IF bComingUp THEN
	IF bEditOffset THEN
		IF bManualPick THEN
			//iCaseRC										:= 900;
			//IF iActualCase = 900 THEN
				bComingUp								:= FALSE;
			//END_IF	
// dodaje druga pozycje pobrania			
		ELSIF bManualPick2 THEN
			//iCaseRC										:= 1600;	
			//IF iActualCase = 1600 THEN
				bComingUp								:= FALSE;
		//	END_IF		
		ELSIF bManualPlace1 THEN
			iCaseRC										:= 1100;	
			IF iActualCase = 1100 THEN
				bComingUp								:= FALSE;
			END_IF	
		ELSIF bManualPlace2 THEN
			iCaseRC										:= 1300;
			//bManualCatch								:= TRUE;
			IF iActualCase = 1300 THEN
				bComingUp								:= FALSE;
			END_IF	
		END_IF	
	ELSE	
		IF iLastCaseRC = 800 THEN												// Pozycja dolna pobierania - komenda
			iCaseRC 										:= 900;
		ELSIF iActualCase = 900 THEN											// Pozycja gorna pobierania - komenda
			iCaseRC											:= 0;
		ELSIF iActualCase = 950 THEN											// Robot w pozycji gornej pobierania
			bComingUp										:= FALSE;
			bManualPick										:= FALSE;			
		ELSIF iLastCaseRC = 1500 THEN											// Pozycja dolna pobierania 2 - komenda
			iCaseRC											:= 1600;
		ELSIF iActualCase = 1600 THEN											// Pozycja gorna pobierania 2 - komenda
			iCaseRC											:= 0;
		ELSIF iActualCase = 1650 THEN											// Robot w pozycji gornej pobierania 2
			bComingUp										:= FALSE;
			bManualPick2									:= FALSE;						
		ELSIF iLastCaseRC = 1000 THEN											// Pozycja dolna odkladania - komenda
			iCaseRC											:= 1100;
		ELSIF iActualCase = 1100 THEN											// Pozycja gorna odkladania - komenda
			iCaseRC											:= 0;
		ELSIF iActualCase = 1150 THEN											// Robot w pozycji gornej odkladania
			bComingUp										:= FALSE;
			bManualPlace1									:= FALSE;
		ELSIF iLastCaseRC = 1200 THEN											// Pozycja dolna odrzutu - komenda
			iCaseRC											:= 1300;
		ELSIF iActualCase = 1300 THEN											// Pozycja gorna odrzutu - komenda
			iCaseRC											:= 0;
		ELSIF iActualCase = 1350 THEN											// Robot w pozycji gornej odrzutu 
			bComingUp										:= FALSE;
			bManualPlace2									:= FALSE;
		END_IF
	END_IF
	iCaseManual												:= 0;	
ELSE
	IF bEditOffset THEN
		IF bManualPick THEN
			iCaseRC											:= 800;				// Pozycja dolna pobierania
		ELSIF bManualPick2 THEN                        	
			iCaseRC											:= 1500;			// Pozycja dolna pobierania 2
		ELSIF bManualPlace1 THEN                        	
			iCaseRC											:= 1000;			// Pozycja dolna odkladanie etykieciarka
		ELSIF bManualPlace2 THEN                        	
			iCaseRC											:= 1200;			// Pozycja dolna odkladania odrzut
		ELSIF iActualCase > 0 THEN                      	
			iCaseRC											:= 0;
		 	bManualPick			:= FALSE;
		 	bManualPick2		:= FALSE;			
		 	bManualPlace1		:= FALSE;
			bManualPlace2		:= FALSE;		
		END_IF	
	iCaseManual												:= 0;	
	ELSE	
//	Case pobranie pojedynczego opakowania	
		IF bManualPick THEN
			CASE iCaseManual OF
				0:
					iCaseRC										:= 200;
					IF iActualCase = 200 THEN
						iCaseRC 								:= 0;
						iCaseManual								:= 10;
					END_IF
				10: 
					IF iActualCase = 250 THEN
						iCaseManual								:= 20;
					END_IF
				20:
					bManualPick									:= FALSE;
					iCaseManual									:= 0;
			END_CASE
		END_IF	
//Dodaje Case bManualPick2 do pobrania dwoch opakowan
		IF bManualPick2 THEN
			CASE iCaseManual OF
				0:
					iCaseRC										:= 1400;
					IF iActualCase = 1400 THEN
						iCaseRC 								:= 0;
						iCaseManual								:= 10;
					END_IF
				10: 
					IF iActualCase = 1450 THEN
						iCaseManual								:= 20;
					END_IF
				20:
					bManualPick2									:= FALSE;
					iCaseManual									:= 0;
			END_CASE
		END_IF		
//	Case odlozenie opakowan na etykieciarke	
		IF bManualPlace1 THEN
			CASE iCaseManual OF
				0:
					iCaseRC										:= 300;
					IF iActualCase = 300 THEN
						iCaseRC 								:= 0;
						iCaseManual								:= 10;
					END_IF
				10: 
					IF iActualCase = 350 THEN
						iCaseManual								:= 20;
					END_IF
				20:
					bManualPlace1								:= FALSE;
					iCaseManual									:= 0;
			END_CASE
		END_IF		
//	Case odlozenie opakowan na odrzut		
		IF bManualPlace2 THEN
			CASE iCaseManual OF
				0:
					iCaseRC										:= 400;
					IF iActualCase = 400 THEN
						iCaseRC 								:= 0;
						iCaseManual								:= 10;
					END_IF
				10: 
					IF iActualCase = 450 THEN
						iCaseManual								:= 20;
					END_IF
				20:
					bManualPlace2								:= FALSE;
					iCaseManual									:= 0;
			END_CASE
		END_IF
//	Case przejazd do pozycji start inkjet		
		IF bManualStartInkJetPosition THEN
			CASE iCaseManual OF
				0:
					iCaseRC										:= 500;
					IF iActualCase = 500 THEN
						iCaseRC 								:= 0;
						iCaseManual								:= 10;
					END_IF
				10: 
					IF iActualCase = 550 THEN
						iCaseManual								:= 20;
					END_IF
				20:
					bManualStartInkJetPosition					:= FALSE;
					iCaseManual									:= 0;
			END_CASE
		END_IF
//	Case przejazd do pozycji stop inkjet		
		IF bManualStopInkJetPosition THEN
			CASE iCaseManual OF
				0:
					iCaseRC										:= 600;
					IF iActualCase = 600 THEN
						iCaseRC 								:= 0;
						iCaseManual								:= 10;
					END_IF
				10: 
					IF iActualCase = 650 THEN
						iCaseManual								:= 20;
					END_IF
				20:
					bManualStopInkJetPosition					:= FALSE;
					iCaseManual									:= 0;
			END_CASE
		END_IF	
		
		IF bManualWeightPosition THEN
			CASE iCaseManual OF
				0:
					iCaseRC										:= 660;
					IF iActualCase = 660 THEN
						iCaseRC 								:= 0;
						iCaseManual								:= 10;
					END_IF
				10: 
					IF iActualCase = 670 THEN
						iCaseManual								:= 20;
					END_IF
				20:	
					iCaseRC										:= 680;
					IF iActualCase = 680 THEN
						iCaseRC 								:= 0;
						iCaseManual								:= 30;
					END_IF	
				30:
					IF iActualCase = 690 THEN
						iCaseManual								:= 40;
					END_IF	
				40:
					bManualWeightPosition						:= FALSE;
					iCaseManual									:= 0;
			END_CASE
		END_IF
		
//	Case przejazd do pozycji gotowosci		
		IF bManualReadyPosition THEN
			CASE iCaseManual OF
				0:
					iCaseRC										:= 700;
					IF iActualCase = 700 THEN
						iCaseRC 								:= 0;
						iCaseManual								:= 10;
					END_IF
				10: 
					IF iActualCase = 750 THEN
						iCaseManual								:= 20;
					END_IF
				20:
					bManualReadyPosition						:= FALSE;
					iCaseManual									:= 0;
			END_CASE
		END_IF	
	END_IF	
END_IF	

IF iCaseRC > 0 THEN
	iLastCaseRC						:= iCaseRC;
END_IF

IF iActualCase=200 OR iActualCase=300 OR iActualCase=400 OR iActualCase=500 OR iActualCase=600 OR iActualCase=700 OR iActualCase=800 OR iActualCase=900 OR iActualCase=1000 OR iActualCase=1100 OR iActualCase=1200 OR iActualCase=1300 OR 
	iActualCase=1400 OR iActualCase=1500 OR iActualCase=1600	THEN
	iBottleTransferLock				:= 2#11111111;	//		nie moge nic
ELSIF iActualCase=150 THEN                                  
	iBottleTransferLock				:= 2#11111110;	//		moge pobrac
ELSIF iActualCase=250 OR iActualCase=950 OR iActualCase=1450 OR iActualCase=1650 THEN	           
	iBottleTransferLock				:= 2#11101001;	//		moge odłozyc, odrzucic i pojechac przed inkjet		
ELSIF iActualCase=350 OR iActualCase=1150 THEN             
	iBottleTransferLock				:= 2#11110111;	//		moge jechac tylko do gotowosci
ELSIF iActualCase=450 OR iActualCase=1350 THEN             
	iBottleTransferLock				:= 2#11110111;	//	   	moge jechac tylko do gotowosci
ELSIF iActualCase=550 THEN                                 
	iBottleTransferLock				:= 2#11011111;	//		moge jechac do koniec inkjet
ELSIF iActualCase=650 THEN                                 
	iBottleTransferLock				:= 2#10101101;	//		moge odłozyc na ety, wrocic przed inkjet
ELSIF iActualCase=750 THEN                                 
	iBottleTransferLock				:= 2#11111110;	//		moge pobrac
END_IF


(*200 pobranie opakowania, 300 odlozenie opakowania, 400 odrzucenie opakowania, 500 przejazd start inkjet, 600 przejazd stop inket, 700 powrot do gotowosci,
800 pozycja dolna pobierania manual, 900 pozycja gorna pobierana manual, 1000 Pozycja dolna odkladania - TRYB MANUALNY, 1100 Pozycja gorna odkladania - TRYB MANUALNY,
1200 Pozycja dolna odrzutu - TRYB MANUALNY, 1300 Pozycja gorna odrzutu - TRYB MANUALNY, 1400 Pobranie  2 opakowan, 1500 Pozycja dolna pobierania 2 - TRYB MANUALNY,
1600 Pozycja gorna pobierania 2 - TRYB MANUALNY


150 - koniec bazowania, 250 - koniec pobierania, 350 - koniec odkladania ety, 450 - koniec odrzutu, 550 - koniec przejazdu do start inket,
650- koniec przejazdu do stop inket, 750 - koniec przejazdu do pozycji gotowosci, 950- koniec gornej pozycji pobrania manual,
1150 - koniec górnej pozycji odkladania manual, 1350 koniec gornej pozycji odrzutu manual, 1450 - koniec pobrania dwoch opakowan,
1650 - koniec gornej pozycji pobrania manual
  *)


(*
IF iActualCase > 0 THEN
	iCaseRC										:= 0;
END_IF
*)
END_ACTION

ACTION Running:
tonWaitForSuckerSensor(IN:=(iActualCase=250 OR iActualCase=350), PT:=T#50MS);

CASE eRunningState OF
  E_RobotMovState.eReadyPlace:	
	iCaseRC								:= 0;
	IF bRun AND NOT bCycleDone THEN
		//Pobór jednego produktu
		IF iPickNumber = 1	THEN
		iCaseRC							:= 200;
			IF iActualCase = 200 THEN
				eRunningState			:= E_RobotMovState.ePicking;
			END_IF
		END_IF
		//Pobor dwóch produktów						
		IF iPickNumber = 2	THEN
		iCaseRC							:= 1400;
			IF iActualCase = 1400 THEN
				eRunningState			:= E_RobotMovState.ePicking;
			END_IF
		END_IF		
		
	END_IF
	
//Sprawdzenie czy poprawnie pobrano produkt
	
	E_RobotMovState.ePicking:
		iCaseRC							:= 0;
		IF  iActualCase = 250 OR iActualLastCase = 250 OR iActualCase = 1450 OR iActualLastCase = 1450 THEN
			iActualLastCase 			:= 0;
			eRunningState				:= E_RobotMovState.ePicked;
		END_IF	

//Sprawdzenie czy popraniw pobrano produkt po zadziałaniu estop	
	E_RobotMovState.ePickingAfterEStop:
		iCaseRC							:= 0;
		IF iActualCase = 280 OR iActualCase = 1480 THEN
			eRunningState				:= E_RobotMovState.ePicked;
		END_IF	
		
// Produkt chwycona do odłożenia 		
	E_RobotMovState.ePicked:
		IF bPlace THEN
			//Odkładanie na etykieciarke
			IF iPlaceNumber = 1 THEN
				IF bInkJetEnable THEN
					iCaseRC				:= 500;
					IF iActualCase = 500 THEN
						eRunningState	:= eMovingInkJetStartPositon;
					END_IF
				ELSE
					iCaseRC				:= 300;
					IF iActualCase = 300 THEN
						eRunningState	:= E_RobotMovState.ePlacing;
					END_IF
				END_IF	
			END_IF
			
			// Odkładanie na odrzut			
			IF iPlaceNumber = 2 THEN
				iCaseRC					:= 400;
				IF iActualCase = 400 THEN
					eRunningState		:= E_RobotMovState.eRejecting;
				END_IF
			END_IF
			
			//Przenoszenie na wagę			
			IF iPlaceNumber = 3 THEN 
				IF bInkJetEnable THEN 
					iCaseRC				:= 500;
					IF iActualCase = 500 THEN
						eRunningState	:= eMovingInkJetStartPositon;
					END_IF
				ELSE
					iCaseRC				:= 660;
					IF iActualCase = 660 THEN
						eRunningState	:= E_RobotMovState.eMovingWeightPosition;
					END_IF
				END_IF	
			END_IF	
			
			
			//Przenoszenie z obrotem
			IF iPlaceNumber = 4 THEN 
				IF bInkJetEnable THEN 
					iCaseRC				:= 500;
					IF iActualCase = 500 THEN
						eRunningState	:= eMovingInkJetStartPositon;
					END_IF
				ELSE
					iCaseRC				:= 1700;
					IF iActualCase = 1700 THEN
						eRunningState	:= E_RobotMovState.eMovingRotatedToPlace;
					END_IF
				END_IF	
			END_IF	
		END_IF		
		
// Sprawdzenie czy odłożono produkt		
	E_RobotMovState.ePlacing:	
		iCaseRC							:= 0;	
		IF iActualCase = 350 THEN
			eRunningState				:= E_RobotMovState.ePlaced;
		END_IF		
		
// Powrót do pozycji gotowości		
	E_RobotMovState.ePlaced:
		iCaseRC							:= 700;
		IF iActualCase = 700 THEN
			eRunningState				:= E_RobotMovState.eReturnToReadyPlace;
		END_IF
		
// Sprawdzenie czy odrzucono produkt		
	E_RobotMovState.eRejecting:
		iCaseRC							:= 0;
		IF iActualCase = 450 THEN	
			eRunningState				:= E_RobotMovState.eRejected;
		END_IF
		
// Sprawdzenie czy odłożono produkt na transporter odrzuconych produktów		
	E_RobotMovState.eRejected:	
		iCaseRC							:= 700;
		IF iActualCase = 700 THEN
			eRunningState				:= E_RobotMovState.eReturnToReadyPlace;
		END_IF
		
// Przejscie do pozycji poczatkowej INKJET		
	E_RobotMovState.eMovingInkJetStartPositon:
		iCaseRC							:= 0;
		IF iActualCase	= 550 THEN
			eRunningState				:= E_RobotMovState.eMovedInkJetStartPositon;
		END_IF
		
// Przejazd INKJET		
	E_RobotMovState.eMovedInkJetStartPositon:
		iCaseRC							:= 600;
		IF iActualCase = 600 THEN
			eRunningState				:= E_RobotMovState.eMovingInkJetStopPositon;
		END_IF	

// Konczenie INJET	
	E_RobotMovState.eMovingInkJetStopPositon:
		iCaseRC							:= 0;	
		IF iActualCase	= 650 THEN
			eRunningState				:= E_RobotMovState.eMovedInkJetStopPositon;
		END_IF	

// Odłożenie opakowania	
	E_RobotMovState.eMovedInkJetStopPositon:
		IF iPlaceNumber = 3 THEN //Przenoszenie na wagę
			iCaseRC				:= 660;
			IF iActualCase = 660 THEN	
				eRunningState	:= eMovingWeightPosition;				
			END_IF 
		ELSE
			iCaseRC							:= 300;	
			IF iActualCase = 300 THEN
				eRunningState				:= E_RobotMovState.ePlacing;
			END_IF	
		END_IF	
	E_RobotMovState.eMovingWeightPosition:
		iCaseRC							:= 0;	
		IF iActualCase = 670 THEN
			eRunningState				:= E_RobotMovState.eMovedWeightPosition;
		END_IF		
	E_RobotMovState.eMovedWeightPosition:
		iCaseRC							:= 680;	
		IF iActualCase = 680 THEN
			eRunningState				:= E_RobotMovState.eMovingAfterWeightPosition;
		END_IF		
	E_RobotMovState.eMovingAfterWeightPosition:
		iCaseRC							:= 0;	
		IF iActualCase = 690 THEN
			eRunningState				:= E_RobotMovState.eMovedAfterWeightPosition;
		END_IF		
	E_RobotMovState.eMovedAfterWeightPosition:
		iCaseRC							:= 300;	
		IF iActualCase = 300 THEN
			eRunningState				:= E_RobotMovState.ePlacing;
		END_IF	
//Odkładanie z obrotem		
	E_RobotMovState.eMovingRotatedToPlace:
		iCaseRC							:= 0;	
		IF iActualCase = 1750 THEN
			eRunningState				:= E_RobotMovState.eReturnToReadyPlace;
		END_IF	
//	E_RobotMovState.eMovedRoatedToPlace:
//		iCaseRC							:= 700;	
//		IF iActualCase = 700 THEN
//			eRunningState				:= E_RobotMovState.eReturnToReadyPlace;
//		END_IF	
		
	
// Konczenie cyklu	
	E_RobotMovState.eReturnToReadyPlace:	
		iCaseRC							:= 0;
		bPlace							:= FALSE;
			//IF iActualCase = 750 THEN
				iLastPickNumber			:= iPlaceNumber;
				bCycleDone				:= TRUE;
			//END_IF
END_CASE

//Tryb wolnych ruchów

IF iPlaceNumber = 1 THEN
	bSlowMotion							:= FALSE;
ELSIF iPlaceNumber = 2 THEN
	bSlowMotion							:= TRUE;	
END_IF
END_ACTION

ACTION Warning:
IF (bEnable) THEN
	
	IF bWarningAcknowledge AND bWarningRCActive  THEN
		bResetWarningRC									:= TRUE;		
	END_IF




	IF bWarningRCActive THEN
		
		bWarning										:= TRUE;
		bWarningNumberRequest							:= TRUE;
		udiWarningId									:= IODATA;
		
		CASE udiWarningId OF	
			
0013:	
	
	sWarningDescription1 := 'Illeagal fileFile Crash';
	sWarningDescription2 := 'File Initial operation';
	
0018:	
	
	sWarningDescription1 := 'The robot model was selected.The robot model was selected.';
	sWarningDescription2 := 'Reset the error';
	
0023:	
	
	sWarningDescription1 := ' Variables save failure (ProgrPower was shutdown before saving program external variables';
	sWarningDescription2 := 'It is necessary to change some parts when not improvement';
	
0024:	
	
	sWarningDescription1 := ' Variables save failure (User)Power was shutdown before saving user-defined external variables';
	sWarningDescription2 := 'The power supply unit might be deteriorated';
	
0029:	
	
	sWarningDescription1 := ' Memory error (ECC)1bit error of ECC was detected';
	sWarningDescription2 := 'When it frequently occurs, contact your service provider';
	
0102:	
	
	sWarningDescription1 := 'Temperature in the Controlle FAN check or Filter at the bottom on Controller becomes old';
	sWarningDescription2 := 'Please exchange the filter to new filter or clean up the filter';
	
0105:	
	
	sWarningDescription1 := ' Temp. in robot CPU is too higAmbient temperature of robot CPU becomes high';
	sWarningDescription2 := 'Please lower ambient temperature to the specification range';
	
0111:	
	
	sWarningDescription1 := ' No UPS battery voltageThe UPS battery is spent';
	sWarningDescription2 := 'Replace the UPS battery';
	
0112:	
	
	sWarningDescription1 := ' Open the UPS battery coverOpen the UPS battery cover';
	sWarningDescription2 := 'Close the UPS battery cover';
	
0114:	
	
	sWarningDescription1 := ' Occur the UPS warningSome abnormalities occurs in UPS';
	sWarningDescription2 := 'Please call S.C.';
	
0120:	
	
	sWarningDescription1 := 'Instantaneous power failureThe power was OFF for 20msec or more';
	sWarningDescription2 := 'Check the power supply connection and power supply state';
	
0150:	
	
	sWarningDescription1 := 'Undefined robot serial numberUndefined robot serial number';
	sWarningDescription2 := 'Input the robot serial number';
	
0151:	
	
	sWarningDescription1 := ' Undefined robot serial numberUndefined robot serial number';
	sWarningDescription2 := 'Input the robot serial number';
	
0152:	
	
	sWarningDescription1 := ' Unmatched robot serial numberRobot arm that connection was replaced';
	sWarningDescription2 := 'Please confirm the connected robot body is not replaced';
	
0190:	
	
	sWarningDescription1 := ' TB not apply present tool No.Connecting TB does not apply present tool number';
	sWarningDescription2 := 'Please operate TB after confirming present tool data(MEXTL)';
	
0200:	
	
	sWarningDescription1 := ' Err.definition file is illegaError number overlapps.';
	sWarningDescription2 := 'Correct Error definition file.';
	
0201:	
	
	sWarningDescription1 := ' Err.definition file is illegaError number is illegal.';
	sWarningDescription2 := 'Correct Error definition file.';
	
0202:	
	
	sWarningDescription1 := ' Err.definition file is illegaError number is out of the range';
	sWarningDescription2 := 'Correct Error definition file.';
	
0203:	
	
	sWarningDescription1 := ' Err.definition file is illegaError definition files form is illegal.';
	sWarningDescription2 := 'Correct Error definition file.';
	
0204:	
	
	sWarningDescription1 := ' Illegal link table was used.System Problem';
	sWarningDescription2 := 'Turn the power OFF and ON once. When it comes back, contact to the dealer.';
	
0205:	
	
	sWarningDescription1 := ' Illegal Error No.System Problem';
	sWarningDescription2 := 'Turn the power OFF and ON once. When it comes back, contact to the dealer.';
	
0240:	
	
	sWarningDescription1 := ' Setting mismatch of safety fuValid/invalid setting of the safety function is a mismatch';
	sWarningDescription2 := 'Turn the power OFF and ON once';
	
0302:	
	
	sWarningDescription1 := ' CR800 test CautionGeneral-purpose Caution for the function test of CR800';
	sWarningDescription2 := 'Check the embedded message';
	
0430:	
	
	sWarningDescription1 := ' Servo amplifier motor overheaThe motor or detectors thermal protector activated';
	sWarningDescription2 := 'Reduce the speed and acceleration of the robot';
	
0460:	
	
	sWarningDescription1 := ' Motor thermal error(Add.Axis)Overheating of the addition axis motor was detected';
	sWarningDescription2 := 'Please exchange the cooling fan of the addition axis motor';
	
1260:	
	
	sWarningDescription1 := 'Encoder communication errorInitial communication error with absolute position linear scale';
	sWarningDescription2 := 'Check the encoder cable connection and conductivity';
	
1270:	
	
	sWarningDescription1 := 'Encoder communication errorThe absolute position serial data was not transmitted correctly';
	sWarningDescription2 := 'Check the encoder cable connection and conductivity';
	
1280:	
	
	sWarningDescription1 := 'Encoder serial format errorAn error was found in the absolute position serial data format';
	sWarningDescription2 := 'Check the encoder cable connection and conductivity';
	
1290:	
	
	sWarningDescription1 := 'Absolute position fluctuationThe absolute position data fluctuated when the power ON';
	sWarningDescription2 := 'Check the axis movement due to arm dropping or external force';
	
1300:	
	
	sWarningDescription1 := 'Servo AMP MP scale F/B errorDeviation was detected in the encoder and MP scale F/B amount';
	sWarningDescription2 := 'Turn the power OFF and ON once';
	
1310:	
	
	sWarningDescription1 := 'Servo AMP MP scale offset errError in the offset data for the ABS position detection system';
	sWarningDescription2 := 'Turn the power OFF and ON once';
	
1320:	
	
	sWarningDescription1 := 'Multi-rotation data errorError was detected in the multi-rotation data for the encoder';
	sWarningDescription2 := 'Turn the power OFF and ON once';
	
1330:	
	
	sWarningDescription1 := 'Encoder battery voltage lowThe voltage of the battery supplying to the encoder has dropped';
	sWarningDescription2 := 'Replace the backup battery';
	
1340:	
	
	sWarningDescription1 := 'Over-regeneration warningThe regeneration level reached 80％ or more';
	sWarningDescription2 := 'Check the load weight or parameter SVPTYP';
	
1350:	
	
	sWarningDescription1 := 'Overload warningThe overload level of servo amplifier reached 80% or more';
	sWarningDescription2 := 'Check the load weight and the robot for collisions, etc';
	
1370:	
	
	sWarningDescription1 := 'Illegal parameter (servo)A parameter was set exceeding the setting range';
	sWarningDescription2 := 'The parameter has not been changed. Reset the correct value';
	
1400:	
	
	sWarningDescription1 := ' regeneration(AUX) frequency oRegeneration at the limit has occurred frequently';
	sWarningDescription2 := 'Check the regeneration capacity';
	
1420:	
	
	sWarningDescription1 := 'Over-regeneration warningThe overload level of converter reached 80% or more';
	sWarningDescription2 := 'Check the load weight or program';
	
1430:	
	
	sWarningDescription1 := 'Servo amplifier main circuit The servo turned ON while the main circuit power was OFF';
	sWarningDescription2 := 'Turn the main circuit power ON';
	
1520:	
	
	sWarningDescription1 := 'Servo motor output watt overThe output wattage of the servo motor exceeded ratings';
	sWarningDescription2 := 'Lower the rotation speed of the servo motor';
	
1580:	
	
	sWarningDescription1 := 'Non-registered servo warningA non-registered servo warning';
	sWarningDescription2 := 'If the warning cannot be reset, turn the power OFF and ON';
	
1620:	
	
	sWarningDescription1 := 'Illegal robot No.The designated robot No. is illegal';
	sWarningDescription2 := 'Set the correct robot No.';
	
1630:	
	
	sWarningDescription1 := 'Cannot servo ON (during errorThe servo cannot be turned ON during a servo error';
	sWarningDescription2 := 'Reset the servo error before turning the servo ON';
	
1650:	
	
	sWarningDescription1 := 'Cannot servo ON (brake OFF)The servo cannot be turned ON when the brakes release';
	sWarningDescription2 := 'Lock the brakes for all axes before turning the servo ON';
	
1660:	
	
	sWarningDescription1 := 'Cannot servo ON (SRVON procesThe servo cannot be turned ON during the servo ON process';
	sWarningDescription2 := 'Do not turn the servo ON during a servo ON process';
	
1670:	
	
	sWarningDescription1 := 'Cannot servo ON (SRVOFF proceThe servo OFF process is being carried out';
	sWarningDescription2 := 'Do not turn the servo OFF during the servo OFF process';
	
1690:	
	
	sWarningDescription1 := 'Cannot brake operation (DEADMThe brakes cannot be released while the DEADMAN switch is OFF';
	sWarningDescription2 := 'Turn the DEADMAN switch ON before operating';
	
1700:	
	
	sWarningDescription1 := 'Cannot brake operation (EMG)The brakes cannot be released while the emergency stop is input';
	sWarningDescription2 := 'Release the emergency stop state before operating';
	
1710:	
	
	sWarningDescription1 := 'Cannot brake operation (SRVONThe brakes cannot be operated during servo ON';
	sWarningDescription2 := 'Turn the servo OFF before operating';
	
1720:	
	
	sWarningDescription1 := 'Cannot brake operation (BRK OThe brakes cannot be released during the brake release process';
	sWarningDescription2 := 'Do not release the brakes during the brake release process';
	
1730:	
	
	sWarningDescription1 := 'Cannot brake operation (BRK OThe brakes cannot be locked during the brake lock process';
	sWarningDescription2 := 'Do not lock the brakes during the brake lock process';
	
1740:	
	
	sWarningDescription1 := 'Servo parameter change failurOther parameter cannot be changed during parameter change';
	sWarningDescription2 := 'Carry out the parameter change process again';
	
1750:	
	
	sWarningDescription1 := 'Servo parameter change failurChanges of the servo parameter failed';
	sWarningDescription2 := 'Carry out the parameter change process again';
	
1760:	
	
	sWarningDescription1 := 'Illegal origin dataThe origin setting data is illegal';
	sWarningDescription2 := 'Set the correct origin data';
	
1761:	
	
	sWarningDescription1 := ' Illegal origin data in robot The origin data is illegal in robot arm';
	sWarningDescription2 := 'Setting the origin';
	
1770:	
	
	sWarningDescription1 := 'Origin setting incompleteThe origin is not set';
	sWarningDescription2 := 'Re-execute after setting the origin';
	
1780:	
	
	sWarningDescription1 := 'Cannot set origin (illegal axThe origin was not set simultaneously for the interference axis';
	sWarningDescription2 := 'Set the origin simultaneously for the interference axis';
	
1781:	
	
	sWarningDescription1 := 'Cannot set origin (SRVON)The origin was set during servo ON';
	sWarningDescription2 := 'Turn the servo OFF before setting the origin';
	
1850:	
	
	sWarningDescription1 := 'Instantaneous power failureThe power was OFF for 20msec or more';
	sWarningDescription2 := 'Check the power supply connection and power supply state';
	
1870:	
	
	sWarningDescription1 := ' Cooling fan stoppedCooling fan in the controller might be out of order';
	sWarningDescription2 := 'Please exchange the cooling fan';
	
1871:	
	
	sWarningDescription1 := 'J1 cooling fan stoppedCooling fan in the controller might be out of order';
	sWarningDescription2 := 'Please exchange the cooling fan';
	
1872:	
	
	sWarningDescription1 := 'J2 cooling fan stoppedCooling fan in the controller might be out of order';
	sWarningDescription2 := 'Please exchange the cooling fan';
	
1873:	
	
	sWarningDescription1 := 'J3 cooling fan stoppedCooling fan in the controller might be out of order';
	sWarningDescription2 := 'Please exchange the cooling fan';
	
1874:	
	
	sWarningDescription1 := 'J4 cooling fan stoppedCooling fan in the controller might be out of order';
	sWarningDescription2 := 'Please exchange the cooling fan';
	
1875:	
	
	sWarningDescription1 := 'J5 cooling fan stoppedCooling fan in the controller might be out of order';
	sWarningDescription2 := 'Please exchange the cooling fan';
	
1876:	
	
	sWarningDescription1 := 'J6 cooling fan stoppedCooling fan in the controller might be out of order';
	sWarningDescription2 := 'Please exchange the cooling fan';
	
1877:	
	
	sWarningDescription1 := 'J7 cooling fan stoppedCooling fan in the controller might be out of order';
	sWarningDescription2 := 'Please exchange the cooling fan';
	
1878:	
	
	sWarningDescription1 := 'J8 cooling fan stoppedCooling fan in the controller might be out of order';
	sWarningDescription2 := 'Please exchange the cooling fan';
	
1890:	
	
	sWarningDescription1 := ' The cooling fan of the additional axis amplifier may be out of order.';
	sWarningDescription2 := '';
	
1891:	
	
	sWarningDescription1 := 'Cooling fan low rev. (add. axCooling fan of the add. axis amp. J1 might be out of order';
	sWarningDescription2 := 'Please exchange the cooling fan';
	
1892:	
	
	sWarningDescription1 := 'Cooling fan low rev. (add. axCooling fan of the add. axis amp. J2 might be out of order';
	sWarningDescription2 := 'Please exchange the cooling fan';
	
1893:	
	
	sWarningDescription1 := 'Cooling fan low rev. (add. axCooling fan of the add. axis amp. J3 might be out of order';
	sWarningDescription2 := 'Please exchange the cooling fan';
	
1894:	
	
	sWarningDescription1 := 'Cooling fan low rev. (add. axCooling fan of the add. axis amp. J4 might be out of order';
	sWarningDescription2 := 'Please exchange the cooling fan';
	
1895:	
	
	sWarningDescription1 := 'Cooling fan low rev. (add. axCooling fan of the add. axis amp. J5 might be out of order';
	sWarningDescription2 := 'Please exchange the cooling fan';
	
1896:	
	
	sWarningDescription1 := 'Cooling fan low rev. (add. axCooling fan of the add. axis amp. J6 might be out of order';
	sWarningDescription2 := 'Please exchange the cooling fan';
	
1897:	
	
	sWarningDescription1 := 'Cooling fan low rev. (add. axCooling fan of the add. axis amp. J7 might be out of order';
	sWarningDescription2 := 'Please exchange the cooling fan';
	
1898:	
	
	sWarningDescription1 := 'Cooling fan low rev. (add. axCooling fan of the add. axis amp. J8 might be out of order';
	sWarningDescription2 := 'Please exchange the cooling fan';
	
1910:	
	
	sWarningDescription1 := 'Cooling fan stopped (amp.)The cooling fan of the servo amp. stopped';
	sWarningDescription2 := 'Confirm the rotation of the servo amp. cooling fan';
	
1920:	
	
	sWarningDescription1 := 'Cooling fan stopped (pow. supThe cooling fan of the power supply stopped';
	sWarningDescription2 := 'Confirm the rotation of the power supply cooling fan';
	
1930:	
	
	sWarningDescription1 := 'Cooling fan stopped (CPU)The cooling fan of the CPU stopped';
	sWarningDescription2 := 'Confirm the rotation of the CPU cooling fan';
	
1940:	
	
	sWarningDescription1 := 'Agitating fan stoppedThe agitating fan in the controller stopped';
	sWarningDescription2 := 'Confirm the rotation of the agitating fan';
	
1960:	
	
	sWarningDescription1 := ' Additional axis AMP warningWarning of the additional axis servo amplifier was detected';
	sWarningDescription2 := 'Please refer to the manual of servo amplifier.';
	
1970:	
	
	sWarningDescription1 := ' Agitating fan stopped (robot)The agitating fan in the robot arm stopped';
	sWarningDescription2 := 'Refer to manual (Troubleshooting)';
	
1990:	
	
	sWarningDescription1 := ' Warning of encoder data errorEncoder positional data error was detected';
	sWarningDescription2 := 'Please check the counter of encoder data error';
	
2040:	
	
	sWarningDescription1 := ' Work coordinate define failedTeaching position is not correct';
	sWarningDescription2 := 'Change the teaching position';
	
2250:	
	
	sWarningDescription1 := ' Safety function is not executSafety function cannot be executed because of origin unsetting';
	sWarningDescription2 := 'Please set the origin';
	
2710:	
	
	sWarningDescription1 := 'CMP error (displacement)The amount of displacement exceeds a regulated value';
	sWarningDescription2 := 'Please reduce displacement';
	
2721:	
	
	sWarningDescription1 := 'CMP error (J1 joint angle)CMP Command exceeds the limit of J1 joint angle';
	sWarningDescription2 := 'Change the position data or reduce displacement';
	
2722:	
	
	sWarningDescription1 := 'CMP error (J2 joint angle)CMP Command exceeds the limit of J2 joint angle';
	sWarningDescription2 := 'Change the position data or reduce displacement';
	
2723:	
	
	sWarningDescription1 := 'CMP error (J3 joint angle)CMP Command exceeds the limit of J3 joint angle';
	sWarningDescription2 := 'Change the position data or reduce displacement';
	
2724:	
	
	sWarningDescription1 := 'CMP error (J4 joint angle)CMP Command exceeds the limit of J4 joint angle';
	sWarningDescription2 := 'Change the position data or reduce displacement';
	
2725:	
	
	sWarningDescription1 := 'CMP error (J5 joint angle)CMP Command exceeds the limit of J5 joint angle';
	sWarningDescription2 := 'Change the position data or reduce displacement';
	
2726:	
	
	sWarningDescription1 := 'CMP error (J6 joint angle)CMP Command exceeds the limit of J6 joint angle';
	sWarningDescription2 := 'Change the position data or reduce displacement';
	
2727:	
	
	sWarningDescription1 := 'CMP error (J7 joint angle)CMP Command exceeds the limit of J7 joint angle';
	sWarningDescription2 := 'Change the position data or reduce displacement';
	
2728:	
	
	sWarningDescription1 := 'CMP error (J8 joint angle)CMP Command exceeds the limit of J8 joint angle';
	sWarningDescription2 := 'Change the position data or reduce displacement';
	
2731:	
	
	sWarningDescription1 := 'CMP error (J1 axis speed)CMP Command exceeds the limit of J1 axis speed';
	sWarningDescription2 := 'Change the position data or reduce the robot motion speed';
	
2732:	
	
	sWarningDescription1 := 'CMP error (J2 axis speed)CMP Command exceeds the limit of J2 axis speed';
	sWarningDescription2 := 'Change the position data or reduce the robot motion speed';
	
2733:	
	
	sWarningDescription1 := 'CMP error (J3 axis speed)CMP Command exceeds the limit of J3 axis speed';
	sWarningDescription2 := 'Change the position data or reduce the robot motion speed';
	
2734:	
	
	sWarningDescription1 := 'CMP error (J4 axis speed)CMP Command exceeds the limit of J4 axis speed';
	sWarningDescription2 := 'Change the position data or reduce the robot motion speed';
	
2735:	
	
	sWarningDescription1 := 'CMP error (J5 axis speed)CMP Command exceeds the limit of J5 axis speed';
	sWarningDescription2 := 'Change the position data or reduce the robot motion speed';
	
2736:	
	
	sWarningDescription1 := 'CMP error (J6 axis speed)CMP Command exceeds the limit of J6 axis speed';
	sWarningDescription2 := 'Change the position data or reduce the robot motion speed';
	
2737:	
	
	sWarningDescription1 := 'CMP error (J7 axis speed)CMP Command exceeds the limit of J7 axis speed';
	sWarningDescription2 := 'Change the position data or reduce the robot motion speed';
	
2738:	
	
	sWarningDescription1 := 'CMP error (J8 axis speed)CMP Command exceeds the limit of J8 axis speed';
	sWarningDescription2 := 'Change the position data or reduce the robot motion speed';
	
2740:	
	
	sWarningDescription1 := 'CMP error (coordinates conv.)CMP Command (POSE type) could not convert to JOINT type';
	sWarningDescription2 := 'Change the position data';
	
2790:	
	
	sWarningDescription1 := ' Cannot teach accurate currentForce control function or CMP command is executed';
	sWarningDescription2 := ' Repeal force control function and compliance mode';
	
3989:	
	
	sWarningDescription1 := ' The test data is undecidedThe tested log data was not decided';
	sWarningDescription2 := 'Please review the argument of the FsTBat command';
	
5610:	
	
	sWarningDescription1 := 'Cannot execute during STOP ONCannot execute during stop signal input';
	sWarningDescription2 := 'Turn the stop signal OFF';
	
5670:	
	
	sWarningDescription1 := ' Cannot execute during waitCannot execute during wait';
	sWarningDescription2 := 'Execute Program Reset';
	
5680:	
	
	sWarningDescription1 := ' Cannot execute while CMP commCannot execute while CMP command is executed';
	sWarningDescription2 := 'Repeal compliance mode (execute CMP OFF)';
	
6050:	
	
	sWarningDescription1 := 'The file cannot be openedMemory size is full';
	sWarningDescription2 := 'Reduce the memory of program size';
	
6060:	
	
	sWarningDescription1 := 'The mode is not TEACHThe mode is not TEACH';
	sWarningDescription2 := 'Carry out parameter writing in the TEACH mode';
	
6070:	
	
	sWarningDescription1 := 'The time cannot be setProgram is runing or robot is SRVON';
	sWarningDescription2 := 'Check the RUN state and that the SRVON state';
	
6080:	
	
	sWarningDescription1 := 'Com mesg is too longCom mesg is too long';
	sWarningDescription2 := 'Check the various settings(ex. Parameters)';
	
6090:	
	
	sWarningDescription1 := 'Can not power reset of robotCan not power reset of robot';
	sWarningDescription2 := 'Can not power reset of robot';
	
6500:	
	
	sWarningDescription1 := 'Not opened COM lineOPEN was not executed by the program';
	sWarningDescription2 := 'Execute OPEN in the program, and then send PRN command';
	
6900:	
	
	sWarningDescription1 := 'Pseudo-input signal modeSet with the parameters';
	sWarningDescription2 := 'When using real signals mode, return the parameter';
	
7000:	
	
	sWarningDescription1 := 'Copy source file was not founThe copy source file was not found';
	sWarningDescription2 := 'Input the correct file name';
	
7010:	
	
	sWarningDescription1 := 'Delete target file was not foThe delete target file was not found';
	sWarningDescription2 := 'Input the correct file name';
	
7020:	
	
	sWarningDescription1 := 'Rename target file was not foThe rename target file was not found';
	sWarningDescription2 := 'Input the correct file name';
	
7040:	
	
	sWarningDescription1 := 'Parameter changes prohibitedChanging this parameter is prohibited as it is dangerous';
	sWarningDescription2 := 'Contact the maker';
	
7070:	
	
	sWarningDescription1 := 'Memory area is fullMemory area is full';
	sWarningDescription2 := 'Delete any unnecessary programs or data';
	
7080:	
	
	sWarningDescription1 := 'Can not read parameterNon-existent parameter or illegal password';
	sWarningDescription2 := '1. Set the correct parameter name. 2. Set the correct password';
	
7081:	
	
	sWarningDescription1 := 'Can not write parameter・Non-existent parameter or illegal password. There are a lot of numbers of characters
							Value is out of range Value is outside the range';
	sWarningDescription2 := '1. Set the correct parameter name. 2. Set the correct password';
	
7082:	
	
	sWarningDescription1 := ' Parameter writing failureFailed in writing the parameter';
	sWarningDescription2 := 'Please confirm a set value and write the parameter again';
	
7090:	
	
	sWarningDescription1 := 'Parameter comment illgalComment illgal';
	sWarningDescription2 := 'Comment is no means.';
	
7110:	
	
	sWarningDescription1 := ' Overhaul period (servo on timThe servo on time has entered the overhaul recommendation period';
	sWarningDescription2 := 'Execution of an overhaul of a robot arm is recommended period';
	
7121:	
	
	sWarningDescription1 := ' Grease replenishment period (Grease consumption degree exceeded the warning level';
	sWarningDescription2 := 'Please replenish grease and reset consumption degree';
	
7122:	
	
	sWarningDescription1 := ' Grease replenishment period (Grease consumption degree exceeded the warning level';
	sWarningDescription2 := 'Please replenish grease and reset consumption degree';
	
7123:	
	
	sWarningDescription1 := ' Grease replenishment period (Grease consumption degree exceeded the warning level';
	sWarningDescription2 := 'Please replenish grease and reset consumption degree';
	
7124:	
	
	sWarningDescription1 := ' Grease replenishment period (Grease consumption degree exceeded the warning level';
	sWarningDescription2 := 'Please replenish grease and reset consumption degree';
	
7125:	
	
	sWarningDescription1 := ' Grease replenishment period (Grease consumption degree exceeded the warning level';
	sWarningDescription2 := 'Please replenish grease and reset consumption degree';
	
7126:	
	
	sWarningDescription1 := ' Grease replenishment period (Grease consumption degree exceeded the warning level';
	sWarningDescription2 := 'Please replenish grease and reset consumption degree';
	
7131:	
	
	sWarningDescription1 := ' Timing belt replacement perioTiming belt consumption degree exceeded the warning level';
	sWarningDescription2 := 'Please replace timing belt and reset consumption degree';
	
7132:	
	
	sWarningDescription1 := ' Timing belt replacement perioTiming belt consumption degree exceeded the warning level';
	sWarningDescription2 := 'Please replace timing belt and reset consumption degree';
	
7133:	
	
	sWarningDescription1 := ' Timing belt replacement perioTiming belt consumption degree exceeded the warning level';
	sWarningDescription2 := 'Please replace timing belt and reset consumption degree';
	
7134:	
	
	sWarningDescription1 := ' Timing belt replacement perioTiming belt consumption degree exceeded the warning level';
	sWarningDescription2 := 'Please replace timing belt and reset consumption degree';
	
7135:	
	
	sWarningDescription1 := ' Timing belt replacement perioTiming belt consumption degree exceeded the warning level';
	sWarningDescription2 := 'Please replace timing belt and reset consumption degree';
	
7136:	
	
	sWarningDescription1 := ' Timing belt replacement perioTiming belt consumption degree exceeded the warning level';
	sWarningDescription2 := 'Please replace timing belt and reset consumption degree';
	
7141:	
	
	sWarningDescription1 := ' Overhaul period (decelerator)Decelerator consumption degree exceeded the warning level';
	sWarningDescription2 := 'Execution of an overhaul of a robot arm is recommended';
	
7142:	
	
	sWarningDescription1 := ' Overhaul period (decelerator)Decelerator consumption degree exceeded the warning level';
	sWarningDescription2 := 'Execution of an overhaul of a robot arm is recommended';
	
7143:	
	
	sWarningDescription1 := ' Overhaul period (decelerator)Decelerator consumption degree exceeded the warning level';
	sWarningDescription2 := 'Execution of an overhaul of a robot arm is recommended';
	
7144:	
	
	sWarningDescription1 := ' Overhaul period (decelerator)Decelerator consumption degree exceeded the warning level';
	sWarningDescription2 := 'Execution of an overhaul of a robot arm is recommended';
	
7145:	
	
	sWarningDescription1 := ' Overhaul period (decelerator)Decelerator consumption degree exceeded the warning level';
	sWarningDescription2 := 'Execution of an overhaul of a robot arm is recommended';
	
7146:	
	
	sWarningDescription1 := ' Overhaul period (decelerator)Decelerator consumption degree exceeded the warning level';
	sWarningDescription2 := 'Execution of an overhaul of a robot arm is recommended';
	
7151:	
	
	sWarningDescription1 := ' Overhaul period (bearing) (J1Bearing consumption degree exceeded the warning level';
	sWarningDescription2 := 'Execution of an overhaul of a robot arm is recommended';
	
7152:	
	
	sWarningDescription1 := ' Overhaul period (bearing) (J2Bearing consumption degree exceeded the warning level';
	sWarningDescription2 := 'Execution of an overhaul of a robot arm is recommended';
	
7153:	
	
	sWarningDescription1 := ' Overhaul period (bearing) (J3Bearing consumption degree exceeded the warning level';
	sWarningDescription2 := 'Execution of an overhaul of a robot arm is recommended';
	
7154:	
	
	sWarningDescription1 := ' Overhaul period (bearing) (J4Bearing consumption degree exceeded the warning level';
	sWarningDescription2 := 'Execution of an overhaul of a robot arm is recommended';
	
7155:	
	
	sWarningDescription1 := ' Overhaul period (bearing) (J5Bearing consumption degree exceeded the warning level';
	sWarningDescription2 := 'Execution of an overhaul of a robot arm is recommended';
	
7156:	
	
	sWarningDescription1 := ' Overhaul period (bearing) (J6Bearing consumption degree exceeded the warning level';
	sWarningDescription2 := 'Execution of an overhaul of a robot arm is recommended';
	
7161:	
	
	sWarningDescription1 := ' Overhaul period (ball screw) Ball screw consumption degree exceeded the war. level';
	sWarningDescription2 := 'Execution of an overhaul of a robot arm is recommended';
	
7162:	
	
	sWarningDescription1 := ' Overhaul period (ball screw) Ball screw consumption degree exceeded the warning level';
	sWarningDescription2 := 'Execution of an overhaul of a robot arm is recommended';
	
7163:	
	
	sWarningDescription1 := ' Overhaul period (ball screw) Ball screw consumption degree exceeded the warning level';
	sWarningDescription2 := 'Execution of an overhaul of a robot arm is recommended';
	
7164:	
	
	sWarningDescription1 := ' Overhaul period (ball screw) Ball screw consumption degree exceeded the warning level';
	sWarningDescription2 := 'Execution of an overhaul of a robot arm is recommended';
	
7165:	
	
	sWarningDescription1 := ' Overhaul period (ball screw) Ball screw consumption degree exceeded the warning level';
	sWarningDescription2 := 'Execution of an overhaul of a robot arm is recommended';
	
7166:	
	
	sWarningDescription1 := ' Overhaul period (ball screw) Ball screw consumption degree exceeded the warning level';
	sWarningDescription2 := 'Execution of an overhaul of a robot arm is recommended';
	
7170:	
	
	sWarningDescription1 := ' Abnormality detection(Dec.)The sign of failure of decelerator was detected';
	sWarningDescription2 := 'Inspection and replacement of decelerator is recommended';
	
7171:	
	
	sWarningDescription1 := ' Abnormality detection(Dec.) (The sign of failure of decelerator was detected';
	sWarningDescription2 := 'Inspection and replacement of decelerator is recommended';
	
7172:	
	
	sWarningDescription1 := ' Abnormality detection(Dec.) (The sign of failure of decelerator was detected';
	sWarningDescription2 := 'Inspection and replacement of decelerator is recommended';
	
7173:	
	
	sWarningDescription1 := ' Abnormality detection(Dec.) (The sign of failure of decelerator was detected';
	sWarningDescription2 := 'Inspection and replacement of decelerator is recommended';
	
7174:	
	
	sWarningDescription1 := ' Abnormality detection(Dec.) (The sign of failure of decelerator was detected';
	sWarningDescription2 := 'Inspection and replacement of decelerator is recommended';
	
7175:	
	
	sWarningDescription1 := ' Abnormality detection(Dec.) (The sign of failure of decelerator was detected';
	sWarningDescription2 := 'Inspection and replacement of decelerator is recommended';
	
7176:	
	
	sWarningDescription1 := ' Abnormality detection(Dec.) (The sign of failure of decelerator was detected';
	sWarningDescription2 := 'Inspection and replacement of decelerator is recommended';
	
7177:	
	
	sWarningDescription1 := ' Abnormality detection(Dec.) (The sign of failure of decelerator was detected';
	sWarningDescription2 := 'Inspection and replacement of decelerator is recommended';
	
7178:	
	
	sWarningDescription1 := ' Abnormality detection(Dec.) (The sign of failure of decelerator was detected';
	sWarningDescription2 := 'Inspection and replacement of decelerator is recommended';
	
7180:	
	
	sWarningDescription1 := ' Abnormality detection(enc datThe sign of failure of encoder was detected';
	sWarningDescription2 := 'Inspection and replacement of motor and wiring is recommended';
	
7181:	
	
	sWarningDescription1 := ' Abnormality detection(enc datThe sign of failure of encoder was detected';
	sWarningDescription2 := 'Inspection and replacement of motor and wiring is recommended';
	
7182:	
	
	sWarningDescription1 := ' Abnormality detection(enc datThe sign of failure of encoder was detected';
	sWarningDescription2 := 'Inspection and replacement of motor and wiring is recommended';
	
7183:	
	
	sWarningDescription1 := ' Abnormality detection(enc datThe sign of failure of encoder was detected';
	sWarningDescription2 := 'Inspection and replacement of motor and wiring is recommended';
	
7184:	
	
	sWarningDescription1 := ' Abnormality detection(enc datThe sign of failure of encoder was detected';
	sWarningDescription2 := 'Inspection and replacement of motor and wiring is recommended';
	
7185:	
	
	sWarningDescription1 := ' Abnormality detection(enc datThe sign of failure of encoder was detected';
	sWarningDescription2 := 'Inspection and replacement of motor and wiring is recommended';
	
7186:	
	
	sWarningDescription1 := ' Abnormality detection(enc datThe sign of failure of encoder was detected';
	sWarningDescription2 := 'Inspection and replacement of motor and wiring is recommended';
	
7187:	
	
	sWarningDescription1 := ' Abnormality detection(enc datThe sign of failure of encoder was detected';
	sWarningDescription2 := 'Inspection and replacement of motor and wiring is recommended';
	
7188:	
	
	sWarningDescription1 := ' Abnormality detection(enc datThe sign of failure of encoder was detected';
	sWarningDescription2 := 'Inspection and replacement of motor and wiring is recommended';
	
7190:	
	
	sWarningDescription1 := ' Abnormality detection(enc comThe sign of failure of encoder was detected';
	sWarningDescription2 := 'Inspection and replacement of motor and wiring is recommended';
	
7191:	
	
	sWarningDescription1 := ' Abnormality detection(enc comThe sign of failure of encoder was detected';
	sWarningDescription2 := 'Inspection and replacement of motor and wiring is recommended';
	
7192:	
	
	sWarningDescription1 := ' Abnormality detection(enc comThe sign of failure of encoder was detected';
	sWarningDescription2 := 'Inspection and replacement of motor and wiring is recommended';
	
7193:	
	
	sWarningDescription1 := ' Abnormality detection(enc comThe sign of failure of encoder was detected';
	sWarningDescription2 := 'Inspection and replacement of motor and wiring is recommended';
	
7194:	
	
	sWarningDescription1 := ' Abnormality detection(enc comThe sign of failure of encoder was detected';
	sWarningDescription2 := 'Inspection and replacement of motor and wiring is recommended';
	
7195:	
	
	sWarningDescription1 := ' Abnormality detection(enc comThe sign of failure of encoder was detected';
	sWarningDescription2 := 'Inspection and replacement of motor and wiring is recommended';
	
7196:	
	
	sWarningDescription1 := ' Abnormality detection(enc comThe sign of failure of encoder was detected';
	sWarningDescription2 := 'Inspection and replacement of motor and wiring is recommended';
	
7197:	
	
	sWarningDescription1 := ' Abnormality detection(enc comThe sign of failure of encoder was detected';
	sWarningDescription2 := 'Inspection and replacement of motor and wiring is recommended';
	
7198:	
	
	sWarningDescription1 := ' Abnormality detection(enc comThe sign of failure of encoder was detected';
	sWarningDescription2 := 'Inspection and replacement of motor and wiring is recommended';
	
7200:	
	
	sWarningDescription1 := ' Add memory has same file.Add memory has file';
	sWarningDescription2 := 'Data clear operation by TB(PROGRAM INIT)';
	
7310:	
	
	sWarningDescription1 := 'Changed variables were not save. The power was OFF during program execution';
	sWarningDescription2 := 'DO NOT turn the power OFF during PROGRAM execution';
	
7320:	
	
	sWarningDescription1 := ' Succeeded in the backup to ROBackup operation was performed';
	sWarningDescription2 := 'As it is, please use it';
	
7321:	
	
	sWarningDescription1 := ' Succeeded in the restore fromAutomatic restoration or compulsive restoration was performed';
	sWarningDescription2 := 'Since ROM data is loaded, please check the contents';
	
7322:	
	
	sWarningDescription1 := ' Failed in the backup to ROMPower supply OFF was carried out during backup processing';
	sWarningDescription2 := 'Please perform backup operation again';
	
7323:	
	
	sWarningDescription1 := ' Failed in the restore from RONone or illegal backup data. or Power supply off of processing';
	sWarningDescription2 := 'Please perform restoration operation again';
	
7324:	
	
	sWarningDescription1 := ' The capacity of ROM and RAM dThere is no extension memory for restoring';
	sWarningDescription2 := 'Please insert an extension memory correctly and perform it again';
	
7410:	
	
	sWarningDescription1 := '1 month inspection is now1 month inspection is now';
	sWarningDescription2 := '1 month inspection is now';
	
7420:	
	
	sWarningDescription1 := '3 month inspection is now3 month inspection is now';
	sWarningDescription2 := '3 month inspection is now';
	
7430:	
	
	sWarningDescription1 := '6 month inspection is now6 month inspection is now';
	sWarningDescription2 := '6 month inspection is now';
	
7440:	
	
	sWarningDescription1 := '1 year inspection is now1 year inspection is now';
	sWarningDescription2 := '1 year inspection is now';
	
7450:	
	
	sWarningDescription1 := 'No battery voltage (robot CPUThe battery is spent';
	sWarningDescription2 := 'Replace the battery and load the data';
	
7451:	
	
	sWarningDescription1 := 'Battery voltage low (robot CPThe battery is spent';
	sWarningDescription2 := 'Replace the battery';
	
7500:	
	
	sWarningDescription1 := 'No battery voltage (robot)The battery is spent';
	sWarningDescription2 := 'Replace the battery and set the origin';
	
7510:	
	
	sWarningDescription1 := 'Battery voltage low (robot)The battery is spent';
	sWarningDescription2 := 'Replace the battery';
	
7520:	
	
	sWarningDescription1 := 'Battery consumption time is oThe battery consumption time was exceeded';
	sWarningDescription2 := 'Replace the battery';
	
7530:	
	
	sWarningDescription1 := 'Replenishment time of greaseIt seems that grease reached longevity';
	sWarningDescription2 := 'Replenish grease';
	
7540:	
	
	sWarningDescription1 := 'Exchange time of the beltIt seems that the belt reached longevity';
	sWarningDescription2 := 'Execute the check and the exchange of the belt';
	
7550:	
	
	sWarningDescription1 := ' Exchange time of the deceleraIt seems that the decelerator reached longevity';
	sWarningDescription2 := 'Execute the check and the exchange of the decelerator';
	
7630:	
	
	sWarningDescription1 := ' No additional-axis cardNo additional-axis card';
	sWarningDescription2 := 'Check additional-axis card';
	
7681:	
	
	sWarningDescription1 := ' Test result was NGThe result of the test processing became NG';
	sWarningDescription2 := 'Please confirm the test object and the test condition';
	
8112:	
	
	sWarningDescription1 := ' ';
	sWarningDescription2 := '';
	
8113:	
	
	sWarningDescription1 := ' ';
	sWarningDescription2 := '';
	
8114:	
	
	sWarningDescription1 := ' ';
	sWarningDescription2 := '';
	
8115:	
	
	sWarningDescription1 := ' ';
	sWarningDescription2 := '';
	
8116:	
	
	sWarningDescription1 := ' ';
	sWarningDescription2 := '';
	
8208:	
	
	sWarningDescription1 := ' There is a possibility of theThe rewriting frequency of ROM exceeded 100000 times';
	sWarningDescription2 := 'Please do not use the trap function';
	
8490:	
	
	sWarningDescription1 := ' DEVICENET Communication test It is communication test mode';
	sWarningDescription2 := 'Please change the mode switch to 3-5 after the test ends';
	
8888:	
	
	sWarningDescription1 := ' Normal Insert-Err MsgNormal Insert-%s-Cause Msg';
	sWarningDescription2 := 'Normal Insert-%s-Measure Msg';
	
8889:	
	
	sWarningDescription1 := ' No InsertMsg-Err MsgNo InsertMsg-Cause Msg';
	sWarningDescription2 := 'No InsertMsg-Measure Msg';
	
8893:	
	
	sWarningDescription1 := ' Get Jiku Nod-Err MsgGet Jiku Nod-Cause Msg';
	sWarningDescription2 := 'Get Jiku Nod Measure Msg';
	
8921:	
	
	sWarningDescription1 := ' Caution of sensor I/F unitThe caution occurred by sensor I/F unit';
	sWarningDescription2 := 'Please refer to the manual of sensor I/F unit';
	
9200:	
	
	sWarningDescription1 := 'User Caution level errorIllegal demand data was transmitted';
	sWarningDescription2 := 'Check program';
	
9201:	
	
	sWarningDescription1 := 'User Caution level errorIllegal demand data was transmitted';
	sWarningDescription2 := 'Check program';
	
9202:	
	
	sWarningDescription1 := 'User Caution level errorIllegal demand data was transmitted';
	sWarningDescription2 := 'Check program';
	
9203:	
	
	sWarningDescription1 := 'User Caution level errorIllegal demand data was transmitted';
	sWarningDescription2 := 'Check program';
	
9204:	
	
	sWarningDescription1 := 'User Caution level errorIllegal demand data was transmitted';
	sWarningDescription2 := 'Check program';
	
9205:	
	
	sWarningDescription1 := 'User Caution level errorIllegal demand data was transmitted';
	sWarningDescription2 := 'Check program';
	
9206:	
	
	sWarningDescription1 := 'User Caution level errorIllegal demand data was transmitted';
	sWarningDescription2 := 'Check program';
	
9207:	
	
	sWarningDescription1 := 'User Caution level errorIllegal demand data was transmitted';
	sWarningDescription2 := 'Check program';
	
9208:	
	
	sWarningDescription1 := 'User Caution level errorIllegal demand data was transmitted';
	sWarningDescription2 := 'Check program';
	
9209:	
	
	sWarningDescription1 := 'User Caution level errorIllegal demand data was transmitted';
	sWarningDescription2 := 'Check program';
	
9210:	
	
	sWarningDescription1 := 'User Caution level errorIllegal demand data was transmitted';
	sWarningDescription2 := 'Check program';
	
9211:	
	
	sWarningDescription1 := 'User Caution level errorIllegal demand data was transmitted';
	sWarningDescription2 := 'Check program';
	
9212:	
	
	sWarningDescription1 := 'User Caution level errorIllegal demand data was transmitted';
	sWarningDescription2 := 'Check program';
	
9213:	
	
	sWarningDescription1 := 'User Caution level errorIllegal demand data was transmitted';
	sWarningDescription2 := 'Check program';
	
9214:	
	
	sWarningDescription1 := 'User Caution level errorIllegal demand data was transmitted';
	sWarningDescription2 := 'Check program';
	
9215:	
	
	sWarningDescription1 := 'User Caution level errorIllegal demand data was transmitted';
	sWarningDescription2 := 'Check program';
	
9216:	
	
	sWarningDescription1 := 'User Caution level errorIllegal demand data was transmitted';
	sWarningDescription2 := 'Check program';
	
9217:	
	
	sWarningDescription1 := 'User Caution level errorIllegal demand data was transmitted';
	sWarningDescription2 := 'Check program';
	
9218:	
	
	sWarningDescription1 := 'User Caution level errorIllegal demand data was transmitted';
	sWarningDescription2 := 'Check program';
	
9219:	
	
	sWarningDescription1 := 'User Caution level errorIllegal demand data was transmitted';
	sWarningDescription2 := 'Check program';
	
9220:	
	
	sWarningDescription1 := 'User Caution level errorIllegal demand data was transmitted';
	sWarningDescription2 := 'Check program';
	
9221:	
	
	sWarningDescription1 := 'User Caution level errorIllegal demand data was transmitted';
	sWarningDescription2 := 'Check program';
	
9222:	
	
	sWarningDescription1 := 'User Caution level errorIllegal demand data was transmitted';
	sWarningDescription2 := 'Check program';
	
9223:	
	
	sWarningDescription1 := 'User Caution level errorIllegal demand data was transmitted';
	sWarningDescription2 := 'Check program';
	
9224:	
	
	sWarningDescription1 := 'User Caution level errorIllegal demand data was transmitted';
	sWarningDescription2 := 'Check program';
	
9225:	
	
	sWarningDescription1 := 'User Caution level errorIllegal demand data was transmitted';
	sWarningDescription2 := 'Check program';
	
9226:	
	
	sWarningDescription1 := 'User Caution level errorIllegal demand data was transmitted';
	sWarningDescription2 := 'Check program';
	
9227:	
	
	sWarningDescription1 := 'User Caution level errorIllegal demand data was transmitted';
	sWarningDescription2 := 'Check program';
	
9228:	
	
	sWarningDescription1 := 'User Caution level errorIllegal demand data was transmitted';
	sWarningDescription2 := 'Check program';
	
9229:	
	
	sWarningDescription1 := 'User Caution level errorIllegal demand data was transmitted';
	sWarningDescription2 := 'Check program';
	
9230:	
	
	sWarningDescription1 := 'User Caution level errorIllegal demand data was transmitted';
	sWarningDescription2 := 'Check program';
	
9231:	
	
	sWarningDescription1 := 'User Caution level errorIllegal demand data was transmitted';
	sWarningDescription2 := 'Check program';
	
9232:	
	
	sWarningDescription1 := 'User Caution level errorIllegal demand data was transmitted';
	sWarningDescription2 := 'Check program';
	
9233:	
	
	sWarningDescription1 := 'User Caution level errorIllegal demand data was transmitted';
	sWarningDescription2 := 'Check program';
	
9234:	
	
	sWarningDescription1 := 'User Caution level errorIllegal demand data was transmitted';
	sWarningDescription2 := 'Check program';
	
9235:	
	
	sWarningDescription1 := 'User Caution level errorIllegal demand data was transmitted';
	sWarningDescription2 := 'Check program';
	
9236:	
	
	sWarningDescription1 := 'User Caution level errorIllegal demand data was transmitted';
	sWarningDescription2 := 'Check program';
	
9237:	
	
	sWarningDescription1 := 'User Caution level errorIllegal demand data was transmitted';
	sWarningDescription2 := 'Check program';
	
9238:	
	
	sWarningDescription1 := 'User Caution level errorIllegal demand data was transmitted';
	sWarningDescription2 := 'Check program';
	
9239:	
	
	sWarningDescription1 := 'User Caution level errorIllegal demand data was transmitted';
	sWarningDescription2 := 'Check program';
	
9240:	
	
	sWarningDescription1 := 'User Caution level errorIllegal demand data was transmitted';
	sWarningDescription2 := 'Check program';
	
9241:	
	
	sWarningDescription1 := 'User Caution level errorIllegal demand data was transmitted';
	sWarningDescription2 := 'Check program';
	
9242:	
	
	sWarningDescription1 := 'User Caution level errorIllegal demand data was transmitted';
	sWarningDescription2 := 'Check program';
	
9243:	
	
	sWarningDescription1 := 'User Caution level errorIllegal demand data was transmitted';
	sWarningDescription2 := 'Check program';
	
9244:	
	
	sWarningDescription1 := 'User Caution level errorIllegal demand data was transmitted';
	sWarningDescription2 := 'Check program';
	
9245:	
	
	sWarningDescription1 := 'User Caution level errorIllegal demand data was transmitted';
	sWarningDescription2 := 'Check program';
	
9246:	
	
	sWarningDescription1 := 'User Caution level errorIllegal demand data was transmitted';
	sWarningDescription2 := 'Check program';
	
9247:	
	
	sWarningDescription1 := 'User Caution level errorIllegal demand data was transmitted';
	sWarningDescription2 := 'Check program';
	
9248:	
	
	sWarningDescription1 := 'User Caution level errorIllegal demand data was transmitted';
	sWarningDescription2 := 'Check program';
	
9249:	
	
	sWarningDescription1 := 'User Caution level errorIllegal demand data was transmitted';
	sWarningDescription2 := 'Check program';
	
9250:	
	
	sWarningDescription1 := 'User Caution level errorIllegal demand data was transmitted';
	sWarningDescription2 := 'Check program';
	
9251:	
	
	sWarningDescription1 := 'User Caution level errorIllegal demand data was transmitted';
	sWarningDescription2 := 'Check program';
	
9252:	
	
	sWarningDescription1 := 'User Caution level errorIllegal demand data was transmitted';
	sWarningDescription2 := 'Check program';
	
9253:	
	
	sWarningDescription1 := 'User Caution level errorIllegal demand data was transmitted';
	sWarningDescription2 := 'Check program';
	
9254:	
	
	sWarningDescription1 := 'User Caution level errorIllegal demand data was transmitted';
	sWarningDescription2 := 'Check program';
	
9255:	
	
	sWarningDescription1 := 'User Caution level errorIllegal demand data was transmitted';
	sWarningDescription2 := 'Check program';
	
9256:	
	
	sWarningDescription1 := 'User Caution level errorIllegal demand data was transmitted';
	sWarningDescription2 := 'Check program';
	
9257:	
	
	sWarningDescription1 := 'User Caution level errorIllegal demand data was transmitted';
	sWarningDescription2 := 'Check program';
	
9258:	
	
	sWarningDescription1 := 'User Caution level errorIllegal demand data was transmitted';
	sWarningDescription2 := 'Check program';
	
9259:	
	
	sWarningDescription1 := 'User Caution level errorIllegal demand data was transmitted';
	sWarningDescription2 := 'Check program';
	
9260:	
	
	sWarningDescription1 := 'User Caution level errorIllegal demand data was transmitted';
	sWarningDescription2 := 'Check program';
	
9261:	
	
	sWarningDescription1 := 'User Caution level errorIllegal demand data was transmitted';
	sWarningDescription2 := 'Check program';
	
9262:	
	
	sWarningDescription1 := 'User Caution level errorIllegal demand data was transmitted';
	sWarningDescription2 := 'Check program';
	
9263:	
	
	sWarningDescription1 := 'User Caution level errorIllegal demand data was transmitted';
	sWarningDescription2 := 'Check program';
	
9264:	
	
	sWarningDescription1 := 'User Caution level errorIllegal demand data was transmitted';
	sWarningDescription2 := 'Check program';
	
9265:	
	
	sWarningDescription1 := 'User Caution level errorIllegal demand data was transmitted';
	sWarningDescription2 := 'Check program';
	
9266:	
	
	sWarningDescription1 := 'User Caution level errorIllegal demand data was transmitted';
	sWarningDescription2 := 'Check program';
	
9267:	
	
	sWarningDescription1 := 'User Caution level errorIllegal demand data was transmitted';
	sWarningDescription2 := 'Check program';
	
9268:	
	
	sWarningDescription1 := 'User Caution level errorIllegal demand data was transmitted';
	sWarningDescription2 := 'Check program';
	
9269:	
	
	sWarningDescription1 := 'User Caution level errorIllegal demand data was transmitted';
	sWarningDescription2 := 'Check program';
	
9270:	
	
	sWarningDescription1 := 'User Caution level errorIllegal demand data was transmitted';
	sWarningDescription2 := 'Check program';
	
9271:	
	
	sWarningDescription1 := 'User Caution level errorIllegal demand data was transmitted';
	sWarningDescription2 := 'Check program';
	
9272:	
	
	sWarningDescription1 := 'User Caution level errorIllegal demand data was transmitted';
	sWarningDescription2 := 'Check program';
	
9273:	
	
	sWarningDescription1 := 'User Caution level errorIllegal demand data was transmitted';
	sWarningDescription2 := 'Check program';
	
9274:	
	
	sWarningDescription1 := 'User Caution level errorIllegal demand data was transmitted';
	sWarningDescription2 := 'Check program';
	
9275:	
	
	sWarningDescription1 := 'User Caution level errorIllegal demand data was transmitted';
	sWarningDescription2 := 'Check program';
	
9276:	
	
	sWarningDescription1 := 'User Caution level errorIllegal demand data was transmitted';
	sWarningDescription2 := 'Check program';
	
9277:	
	
	sWarningDescription1 := 'User Caution level errorIllegal demand data was transmitted';
	sWarningDescription2 := 'Check program';
	
9278:	
	
	sWarningDescription1 := 'User Caution level errorIllegal demand data was transmitted';
	sWarningDescription2 := 'Check program';
	
9279:	
	
	sWarningDescription1 := 'User Caution level errorIllegal demand data was transmitted';
	sWarningDescription2 := 'Check program';
	
9280:	
	
	sWarningDescription1 := 'User Caution level errorIllegal demand data was transmitted';
	sWarningDescription2 := 'Check program';
	
9281:	
	
	sWarningDescription1 := 'User Caution level errorIllegal demand data was transmitted';
	sWarningDescription2 := 'Check program';
	
9282:	
	
	sWarningDescription1 := 'User Caution level errorIllegal demand data was transmitted';
	sWarningDescription2 := 'Check program';
	
9283:	
	
	sWarningDescription1 := 'User Caution level errorIllegal demand data was transmitted';
	sWarningDescription2 := 'Check program';
	
9284:	
	
	sWarningDescription1 := 'User Caution level errorIllegal demand data was transmitted';
	sWarningDescription2 := 'Check program';
	
9285:	
	
	sWarningDescription1 := 'User Caution level errorIllegal demand data was transmitted';
	sWarningDescription2 := 'Check program';
	
9286:	
	
	sWarningDescription1 := 'User Caution level errorIllegal demand data was transmitted';
	sWarningDescription2 := 'Check program';
	
9287:	
	
	sWarningDescription1 := 'User Caution level errorIllegal demand data was transmitted';
	sWarningDescription2 := 'Check program';
	
9288:	
	
	sWarningDescription1 := 'User Caution level errorIllegal demand data was transmitted';
	sWarningDescription2 := 'Check program';
	
9289:	
	
	sWarningDescription1 := 'User Caution level errorIllegal demand data was transmitted';
	sWarningDescription2 := 'Check program';
	
9290:	
	
	sWarningDescription1 := 'User Caution level errorIllegal demand data was transmitted';
	sWarningDescription2 := 'Check program';
	
9291:	
	
	sWarningDescription1 := 'User Caution level errorIllegal demand data was transmitted';
	sWarningDescription2 := 'Check program';
	
9292:	
	
	sWarningDescription1 := 'User Caution level errorIllegal demand data was transmitted';
	sWarningDescription2 := 'Check program';
	
9293:	
	
	sWarningDescription1 := 'User Caution level errorIllegal demand data was transmitted';
	sWarningDescription2 := 'Check program';
	
9294:	
	
	sWarningDescription1 := 'User Caution level errorIllegal demand data was transmitted';
	sWarningDescription2 := 'Check program';
	
9295:	
	
	sWarningDescription1 := 'User Caution level errorIllegal demand data was transmitted';
	sWarningDescription2 := 'Check program';
	
9296:	
	
	sWarningDescription1 := 'User Caution level errorIllegal demand data was transmitted';
	sWarningDescription2 := 'Check program';
	
9297:	
	
	sWarningDescription1 := 'User Caution level errorIllegal demand data was transmitted';
	sWarningDescription2 := 'Check program';
	
9298:	
	
	sWarningDescription1 := 'User Caution level errorIllegal demand data was transmitted';
	sWarningDescription2 := 'Check program';
	
9299:	
	
	sWarningDescription1 := 'User Caution level errorIllegal demand data was transmitted';
	sWarningDescription2 := 'Check program';

			
		END_CASE
		
	ELSE
	bWarningNumberRequest									:= FALSE;
	bResetWarningRC											:= FALSE;	
	bWarning												:= FALSE;
	sWarningDescription1									:= '';
	sWarningDescription2 									:= ''; 
	
	END_IF
	
ELSE
	udiWarningId											:= 0;
	bWarning												:= 	FALSE;
	sWarningDescription1									:= '';
	sWarningDescription2 									:= ''; 
		
END_IF
END_ACTION

END_FUNCTION_BLOCK

// ---- POUs/FB/Conversions/FB_IntTo2Byte.TcPOU
(****************************************************************************************)
(*							Beckhoff Automation Poland									*)
(*								FB_IntTo2Byte	 v1.0									*)
(*									24.5.2011											*)
(*			Blok funkcyjny rozbijający zmienną typu INT na dwie zmienne typu BYTE		*)
(*______________________________________________________________________________________*)
FUNCTION_BLOCK FB_IntTo2Byte
VAR_INPUT
	iInput :INT;
END_VAR
VAR_OUTPUT
	byStarszy : BYTE;
	byMlodszy : BYTE;
END_VAR

byMlodszy := INT_TO_BYTE(iInput);
byStarszy := INT_TO_BYTE(ROL(iInput, 8));

END_FUNCTION_BLOCK

// ---- POUs/P01_TwoPhasesBarriers.TcPOU
PROGRAM P01_TwoPhasesBarriers
VAR_INPUT
IbBarrierBetweenWeightOpenedSensor 			AT %I*: BOOL;	
IbBarrierBetweenWeightClosedSensor 			AT %I*: BOOL;
IbBarrierBetweenDispencerOpenedSensor 		AT %I*: BOOL;
IbBarrierBetweenDispencerClosedSensor 		AT %I*: BOOL;
IbGateBeforeWeights56				 		AT %I*: BOOL;
END_VAR



VAR
	
	QbBarrierBetweenDispencerActuator 			: BOOL; 				 // Wyjście sterujące szlabanem ruchomym pod dozownikami
	//IbBarrierBetweenDispencerOpenedSensor 		AT %I*: BOOL; 			 // Wejście czujnika siłownika środkowej ruchomej bandy pod dozownikami
	//IbBarrierBetweenDispencerClosedSensor 		AT %I*: BOOL; 			 // Wejście czujnika siłownika środkowej ruchomej bandy pod dozownikami

	QbBarrierBetweenWeightActuator 			: BOOL; 				 // Wyjście sterujące szlabanem przed wagami
	
	//IbBarrierBetweenWeightOpenedSensor 			AT %I*: BOOL; 			// Wejście czujnika siłownika środkowej ruchomej bandy przed wjazdem na wagę
	//IbBarrierBetweenWeightClosedSensor 			AT %I*: BOOL; 			// Wejście czujnika siłownika środkowej ruchomej bandy przed wjazdem na wagę

	
	fbBarrierDispencer							: FB_Gate;				// Bloczek obsługi bandy 
	fbBarrierWeight								: FB_Gate;				// Bloczek obsługi bandy 	
	
	bTemp: BOOL;
END_VAR

aBeforeWeight();
aBetweenDispencer();

ACTION aBeforeWeight:
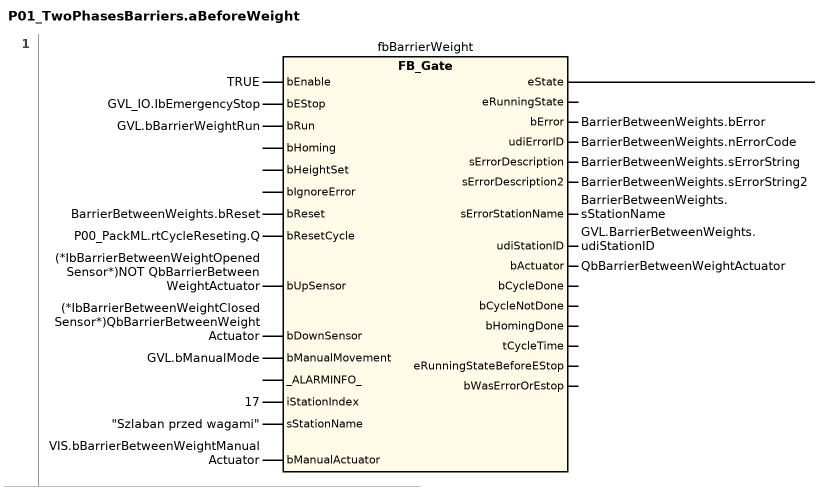
// NETWORK 1
fbBarrierWeight(
    bEnable := TRUE,
    bEStop := GVL_IO.IbEmergencyStop,
    bRun := GVL.bBarrierWeightRun,
    bReset := BarrierBetweenWeights.bReset,
    bResetCycle := P00_PackML.rtCycleReseting.Q,
    bUpSensor := (*IbBarrierBetweenWeightOpenedSensor*)NOT QbBarrierBetweenWeightActuator,
    bDownSensor := (*IbBarrierBetweenWeightClosedSensor*)QbBarrierBetweenWeightActuator,
    bManualMovement := GVL.bManualMode,
    iStationIndex := 17,
    sStationName := "Szlaban przed wagami",
    bManualActuator := VIS.bBarrierBetweenWeightManualActuator,
    bError => BarrierBetweenWeights.bError,
    udiErrorID => BarrierBetweenWeights.nErrorCode,
    sErrorDescription => BarrierBetweenWeights.sErrorString,
    sErrorDescription2 => BarrierBetweenWeights.sErrorString2,
    sErrorStationName => BarrierBetweenWeights.sStationName,
    udiStationID => GVL.BarrierBetweenWeights.udiStationID,
    bActuator => QbBarrierBetweenWeightActuator); // FB_Gate
END_ACTION

ACTION aBetweenDispencer:
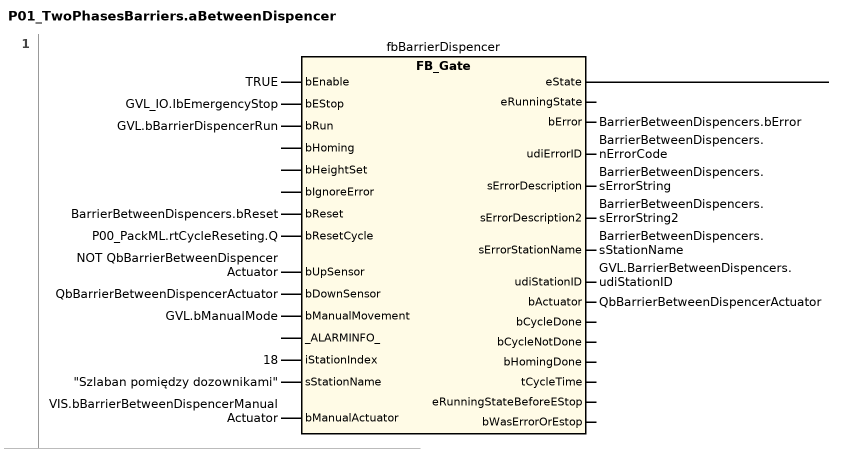
// NETWORK 1
fbBarrierDispencer(
    bEnable := TRUE,
    bEStop := GVL_IO.IbEmergencyStop,
    bRun := GVL.bBarrierDispencerRun,
    bReset := BarrierBetweenDispencers.bReset,
    bResetCycle := P00_PackML.rtCycleReseting.Q,
    bUpSensor := NOT QbBarrierBetweenDispencerActuator,
    bDownSensor := QbBarrierBetweenDispencerActuator,
    bManualMovement := GVL.bManualMode,
    iStationIndex := 18,
    sStationName := "Szlaban pomiędzy dozownikami",
    bManualActuator := VIS.bBarrierBetweenDispencerManualActuator,
    bError => BarrierBetweenDispencers.bError,
    udiErrorID => BarrierBetweenDispencers.nErrorCode,
    sErrorDescription => BarrierBetweenDispencers.sErrorString,
    sErrorDescription2 => BarrierBetweenDispencers.sErrorString2,
    sErrorStationName => BarrierBetweenDispencers.sStationName,
    udiStationID => GVL.BarrierBetweenDispencers.udiStationID,
    bActuator => QbBarrierBetweenDispencerActuator); // FB_Gate
END_ACTION

END_PROGRAM

// ---- POUs/P01_Gates.TcPOU
PROGRAM P01_Gates
VAR_INPUT
	IbGateBeforeWeight14AfterSensor					:BOOL;
	IbLidFeederBarrierOnSensor 	AT %I*  : BOOL;		
    IbLidFeederBarrierOffSensor AT %I*  : BOOL;		
	IbGateBeforeWeights14Sensor	AT %I*	:BOOL;	
	IbGateBeforeWeights56Sensor	AT %I*	:BOOL;		 
END_VAR

VAR
//Szlaban przed dozownikami
	fbGateBeforeDispencers: FB_SpringGateV2;
	fbGateBeforeDispencersState: FB_State;
	eGateBeforeDispencersState :E_Station;
	eGateBeforeDispencersRunningState:E_EntranceGatesState; 
	
	tofTimerGateBeforeDispencersEnable: TOF;
	QbGateBeforeDispencersActuator : BOOL; 				 // Wyjście sterujące szlabanem nr 1 pod robotem
	QbGate0BeforeDispencersActuator : BOOL; 				// Wyjście sterujące szlabanem nr 1 pod robotem
	
//Szlabany przed wagami
	QbGateBeforeWeight14Actuator : BOOL; 			
	QbGateBeforeWeight56Actuator : BOOL; 		

// Szlaban pod stacja robota
	fbGateRobot: FB_SpringGateV2;
	fbGateRobotState: FB_State;
	eGateRobotState :E_Station;
	eGateRobotRunningState:E_EntranceGatesState; 
	tofTimerBottleTransferGatesEnable: TOF;

	QbBottleTransferGate1Actuator : BOOL; 			(*od robota*)	 // Wyjście sterujące szlabanem nr 1 pod robotem
	
	
	fbLidFeederBarrier: FB_Gate;
	QbLidFeederBarrierActuator : BOOL; 	
				
		
	
END_VAR

{warning 'Oprogramować szlaban 0 którego nie było'}
QbGate0BeforeDispencersActuator := QbGateBeforeDispencersActuator;

aGateBeforeDispencers();
aGateBeforeWeight();
aGateRobot();
aLidFeederBarrier();

(***** Generowanie stanu stacji do wizki***********)

//Stan szlabanu przed dozownikami
fbGateBeforeDispencersState(
	eState:= eGateBeforeDispencersState, 
	bRun:=VIS.bGateBeforeDispencersRun AND NOT bManualMode,
	eEntranceGatesRunningState:= eGateBeforeDispencersRunningState, 
	sStateDesc=> VIS.sGateBeforeDispencersState,
	iState=>VIS.iGateBeforeDispencersState);	

(*Opoznienie wyłączanie enabla*)
tofTimerGateBeforeDispencersEnable (IN:=bGateBeforeDispencersEnable , PT:=T#2S);
(*
//Stan szlabanu za wagami
fbGateAfterWeightState(
	eState:= eGateAfterWeightState, 
	bRun:=VIS.bGateAfterWeightEntranceRun AND NOT bManualMode,
	eEntranceGatesRunningState:= eGateAfterWeightRunningState, 
	sStateDesc=> VIS.sGateAfterWeightState,
	iState=>VIS.iGateAfterWeightState);	
*)	
IF P00_PackML.fbPMLAuto.ePMLState = E_PMLState.ePMLState_IDLE THEN
	nGateAfterWeightTimeFormInserting:=250;
END_IF

//Stan szlabanu pod robotem
fbGateRobotState(
	eState:= eGateRobotState, 
	bRun:=VIS.bGateRobotEntranceRun AND NOT bManualMode,
	eEntranceGatesRunningState:= eGateRobotRunningState, 
	sStateDesc=> VIS.sGateRobotState,
	iState=>VIS.iGateRobotState);	
	
IF P00_PackML.fbPMLAuto.ePMLState = E_PMLState.ePMLState_IDLE THEN
	GVL.nGateRobotTimeFormInserting:=250;
END_IF

(*Opoznienie wyłączanie enabla*)
tofTimerBottleTransferGatesEnable (IN:=GVL.bGateRobotEnable , PT:=T#2S);

ACTION aGateBeforeDispencers:
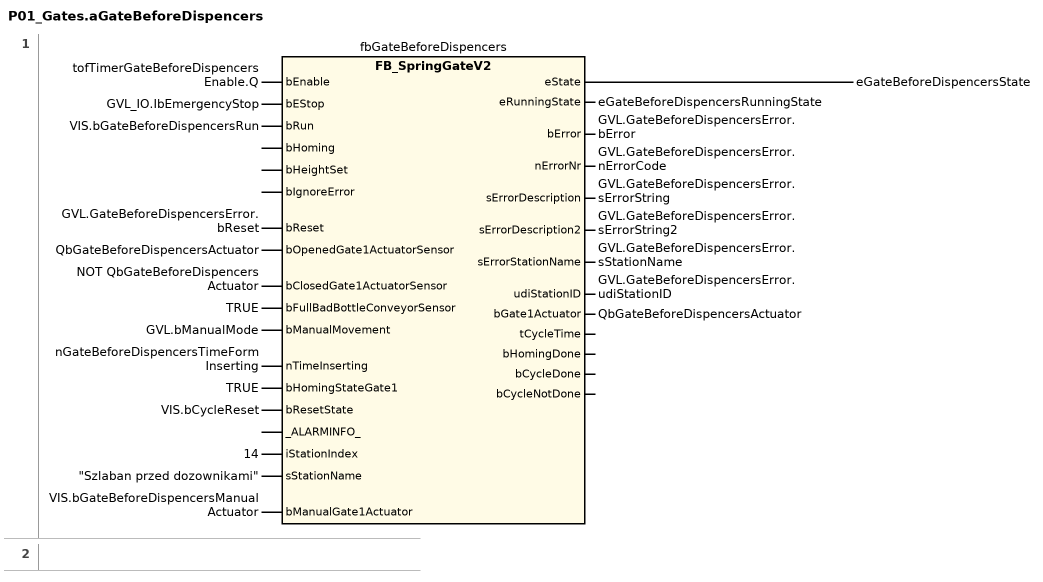
// NETWORK 1
fbGateBeforeDispencers(
    bEnable := tofTimerGateBeforeDispencersEnable.Q,
    bEStop := GVL_IO.IbEmergencyStop,
    bRun := VIS.bGateBeforeDispencersRun,
    bReset := GVL.GateBeforeDispencersError.bReset,
    bOpenedGate1ActuatorSensor := QbGateBeforeDispencersActuator,
    bClosedGate1ActuatorSensor := NOT QbGateBeforeDispencersActuator,
    bFullBadBottleConveyorSensor := TRUE,
    bManualMovement := GVL.bManualMode,
    nTimeInserting := nGateBeforeDispencersTimeFormInserting,
    bHomingStateGate1 := TRUE,
    bResetState := VIS.bCycleReset,
    iStationIndex := 14,
    sStationName := "Szlaban przed dozownikami",
    bManualGate1Actuator := VIS.bGateBeforeDispencersManualActuator,
    eRunningState => eGateBeforeDispencersRunningState,
    bError => GVL.GateBeforeDispencersError.bError,
    nErrorNr => GVL.GateBeforeDispencersError.nErrorCode,
    sErrorDescription => GVL.GateBeforeDispencersError.sErrorString,
    sErrorDescription2 => GVL.GateBeforeDispencersError.sErrorString2,
    sErrorStationName => GVL.GateBeforeDispencersError.sStationName,
    udiStationID => GVL.GateBeforeDispencersError.udiStationID,
    bGate1Actuator => QbGateBeforeDispencersActuator); // FB_SpringGateV2
eGateBeforeDispencersState := fbGateBeforeDispencers.eState;

// NETWORK 2
END_ACTION

ACTION aGateBeforeWeight:

QbGateBeforeWeight14Actuator := VIS.bGateBeforeWeight14Run ;
VIS.bGateBeforeWeight14ManualActuator;

QbGateBeforeWeight56Actuator := VIS.bGateBeforeWeight56Run ;
VIS.bGateBeforeWeight56ManualActuator;
END_ACTION

ACTION aGateRobot:
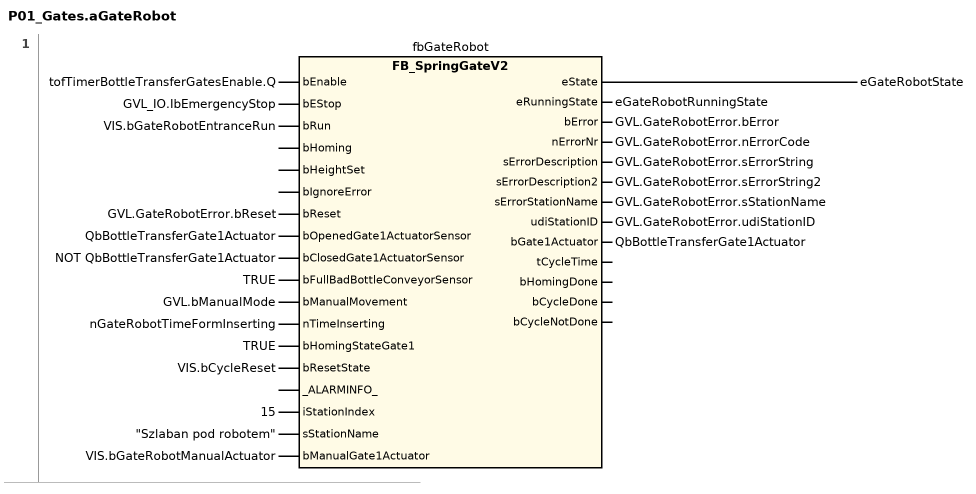
// NETWORK 1
fbGateRobot(
    bEnable := tofTimerBottleTransferGatesEnable.Q,
    bEStop := GVL_IO.IbEmergencyStop,
    bRun := VIS.bGateRobotEntranceRun,
    bReset := GVL.GateRobotError.bReset,
    bOpenedGate1ActuatorSensor := QbBottleTransferGate1Actuator,
    bClosedGate1ActuatorSensor := NOT QbBottleTransferGate1Actuator,
    bFullBadBottleConveyorSensor := TRUE,
    bManualMovement := GVL.bManualMode,
    nTimeInserting := nGateRobotTimeFormInserting,
    bHomingStateGate1 := TRUE,
    bResetState := VIS.bCycleReset,
    iStationIndex := 15,
    sStationName := "Szlaban pod robotem",
    bManualGate1Actuator := VIS.bGateRobotManualActuator,
    eRunningState => eGateRobotRunningState,
    bError => GVL.GateRobotError.bError,
    nErrorNr => GVL.GateRobotError.nErrorCode,
    sErrorDescription => GVL.GateRobotError.sErrorString,
    sErrorDescription2 => GVL.GateRobotError.sErrorString2,
    sErrorStationName => GVL.GateRobotError.sStationName,
    udiStationID => GVL.GateRobotError.udiStationID,
    bGate1Actuator => QbBottleTransferGate1Actuator); // FB_SpringGateV2
eGateRobotState := fbGateRobot.eState;
END_ACTION

ACTION aLidFeederBarrier:
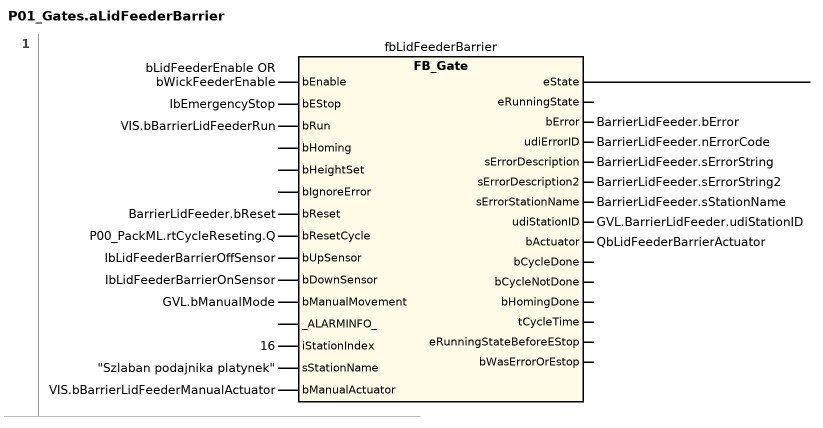
// NETWORK 1
fbLidFeederBarrier(
    bEnable := bLidFeederEnable OR bWickFeederEnable,
    bEStop := IbEmergencyStop,
    bRun := VIS.bBarrierLidFeederRun,
    bReset := BarrierLidFeeder.bReset,
    bResetCycle := P00_PackML.rtCycleReseting.Q,
    bUpSensor := IbLidFeederBarrierOffSensor,
    bDownSensor := IbLidFeederBarrierOnSensor,
    bManualMovement := GVL.bManualMode,
    iStationIndex := 16,
    sStationName := "Szlaban podajnika platynek",
    bManualActuator := VIS.bBarrierLidFeederManualActuator,
    bError => BarrierLidFeeder.bError,
    udiErrorID => BarrierLidFeeder.nErrorCode,
    sErrorDescription => BarrierLidFeeder.sErrorString,
    sErrorDescription2 => BarrierLidFeeder.sErrorString2,
    sErrorStationName => BarrierLidFeeder.sStationName,
    udiStationID => GVL.BarrierLidFeeder.udiStationID,
    bActuator => QbLidFeederBarrierActuator); // FB_Gate
END_ACTION

END_PROGRAM

// ---- POUs/P05_Weight.TcPOU
(*
Nazwa:			P05_Weight
Opis:			Stacja wagi
Wersja:			v0.2
Data:			2019-10-1
Autor:			DP
Urzadzenia:		
Konfiguracja:	
Info:
-przerobione na wagę beckhofa
*)
PROGRAM P05_Weight
VAR_INPUT
	IbWeight1FormSensor						AT %I*		: BOOL;							//Czujnik nad Waga 1
	IbWeight2FormSensor						AT %I*		: BOOL;							//Czujnik nad Waga 2
	IbWeight3FormSensor						AT %I*		: BOOL;							//Czujnik nad Waga 3
	IbWeight4FormSensor						AT %I*		: BOOL;							//Czujnik nad Waga 4
	IbWeight5FormSensor						AT %I*		: BOOL;							//Czujnik nad Waga 4
	IbWeight6FormSensor						AT %I*		: BOOL;							//Czujnik nad Waga 4
END_VAR
VAR
	//Podnosnik szalek
	
	//eWeightLiftRunningState			:E_WeightLiftState;				// Stan pracy podajnika
	fbWeightLiftState					:FB_State;
	
	//Waga 1
	fbWeight1							:FB_BeckhoffEL3356Weight;		// Blok sterujący pierwszą wagą
	eWeight1State						:E_Station; 					// Stan pracy podajnika platynek			
	eWeight1RunningState				:E_WeightState; 				// Stan pracy podajnika platynek
	fbWeight1State						:FB_State;					

	(*No nowej wagi*)
	(*wejścia*)
	InWeight1Value						 AT %I*: DINT;			// Wartość wagi
	IbWeight1Overrange					 AT %I*: BOOL;						
	IbWeight1DataInvalid				 AT %I*: BOOL;		
	IbWeight1Error 						 AT %I*: BOOL;	
	IbWeight1CalibrationInProgress 		 AT %I*: BOOL;
	IbWeight1SteadyState				 AT %I*: BOOL;
	IbWeight1SyncError 					 AT %I*: BOOL;
	(*wyjścia*)
	QbWeight1StartCalibration 			 AT %Q*: BOOL;
	QbWeight1DisableCalibration     	 AT %Q*: BOOL;
	QbWeight1InputFreeze 				 AT %Q*: BOOL;
	QbWeight1SampleMode 				 AT %Q*: BOOL;
	QbWeight1Tara 					     AT %Q*: BOOL;
	
	(*Ostrzezenia*)
	bWeight1Warning1					:BOOL; // 
	tonWeight1Tare						:TON;
	
	//Waga 2
	fbWeight2							:FB_BeckhoffEL3356Weight;		// Blok sterujący pierwszą wagą
	eWeight2State						:E_Station; 					// Stan pracy podajnika platynek			
	eWeight2RunningState				:E_WeightState; 				// Stan pracy podajnika platynek
	fbWeight2State						:FB_State;					

	(*No nowej wagi*)
	(*wejścia*)
	InWeight2Value 						AT %I*: DINT;			// Wartość wagi
	IbWeight2Overrange 					AT %I*: BOOL;						
	IbWeight2DataInvalid 				AT %I*: BOOL;		
	IbWeight2Error 						AT %I*: BOOL;	
	IbWeight2CalibrationInProgress		AT %I*: BOOL;
	IbWeight2SteadyState 				AT %I*: BOOL;
	IbWeight2SyncError 					AT %I*: BOOL;
	(*wyjścia*)
	QbWeight2StartCalibration 			AT %Q*: BOOL;
	QbWeight2DisableCalibration			AT %Q*: BOOL;
	QbWeight2InputFreeze 				AT %Q*: BOOL;
	QbWeight2SampleMode 				AT %Q*: BOOL;
	QbWeight2Tara 						AT %Q*: BOOL;
	
	(*Ostrzezenia*)
	bWeight2Warning1					:BOOL; // 
	tonWeight2Tare						:TON;
		
	//Waga 3
	fbWeight3							:FB_BeckhoffEL3356Weight;		// Blok sterujący pierwszą wagą
	eWeight3State						:E_Station; 					// Stan pracy podajnika platynek			
	eWeight3RunningState				:E_WeightState; 				// Stan pracy podajnika platynek
	fbWeight3State						:FB_State;					

	(*No nowej wagi*)
	(*wejścia*)
	InWeight3Value						 AT %I*: DINT;			// Wartość wagi
	IbWeight3Overrange 					 AT %I*: BOOL;						
	IbWeight3DataInvalid 				 AT %I*: BOOL;		
	IbWeight3Error 						 AT %I*: BOOL;	
	IbWeight3CalibrationInProgress 		 AT %I*: BOOL;
	IbWeight3SteadyState 				 AT %I*: BOOL;
	IbWeight3SyncError 					 AT %I*: BOOL;
	(*wyjścia*)
	QbWeight3StartCalibration 			 AT %Q*: BOOL;
	QbWeight3DisableCalibration 		 AT %Q*: BOOL;
	QbWeight3InputFreeze 				 AT %Q*: BOOL;
	QbWeight3SampleMode 			   	 AT %Q*: BOOL;
	QbWeight3Tara 						 AT %Q*: BOOL;
	
	(*Ostrzezenia*)
	bWeight3Warning1					:BOOL; // 
	tonWeight3Tare						: TON;	
	
	//Waga 4
	fbWeight4							:FB_BeckhoffEL3356Weight;		// Blok sterujący pierwszą wagą
	eWeight4State						:E_Station; 					// Stan pracy podajnika platynek			
	eWeight4RunningState				:E_WeightState; 				// Stan pracy podajnika platynek
	fbWeight4State						:FB_State;					

	(*No nowej wagi*)
	(*wejścia*)
	InWeight4Value 						AT %I*: DINT;			// Wartość wagi
	IbWeight4Overrange 					AT %I*: BOOL;						
	IbWeight4DataInvalid				AT %I*: BOOL;		
	IbWeight4Error 						AT %I*: BOOL;	
	IbWeight4CalibrationInProgress 		AT %I*: BOOL;
	IbWeight4SteadyState 				AT %I*: BOOL;
	IbWeight4SyncError 					AT %I*: BOOL;
	(*wyjścia*)
	QbWeight4StartCalibration 			AT %Q*: BOOL;
	QbWeight4DisableCalibration 		AT %Q*: BOOL;
	QbWeight4InputFreeze 				AT %Q*: BOOL;
	QbWeight4SampleMode 				AT %Q*: BOOL;
	QbWeight4Tara 						AT %Q*: BOOL;

	(*Ostrzezenia*)
	bWeight4Warning1					:BOOL; // 
	tonWeight4Tare						:TON;	
		
(******** Dozowanie dwufazowe******)	
////// Wagi przy dozowaniu dwufazowym dodano 07.04.2022
	//Waga 5
	fbWeight5							:FB_BeckhoffEL3356Weight;		// Blok sterujący pierwszą wagą
	eWeight5State						:E_Station; 					// Stan pracy podajnika platynek			
	eWeight5RunningState				:E_WeightState; 				// Stan pracy podajnika platynek
	fbWeight5State						:FB_State;					

	(*No nowej wagi*)
	(*wejścia*)
	InWeight5Value 						AT %I*: DINT;			// Wartość wagi
	IbWeight5Overrange 					AT %I*: BOOL;						
	IbWeight5DataInvalid 				AT %I*: BOOL;		
	IbWeight5Error 						AT %I*: BOOL;	
	IbWeight5CalibrationInProgress 		AT %I*: BOOL;
	IbWeight5SteadyState 				AT %I*: BOOL;
	IbWeight5SyncError 					AT %I*: BOOL;
	(*wyjścia*)
	QbWeight5StartCalibration 			AT %Q*: BOOL;
	QbWeight5DisableCalibration 		AT %Q*: BOOL;
	QbWeight5InputFreeze 				AT %Q*: BOOL;
	QbWeight5SampleMode 				AT %Q*: BOOL;
	QbWeight5Tara 						AT %Q*: BOOL;

	(*Ostrzezenia*)
	bWeight5Warning1					:BOOL; // 
	tonWeight5Tare						:TON;		
	
	//Waga 5
	fbWeight6							:FB_BeckhoffEL3356Weight;		// Blok sterujący pierwszą wagą
	eWeight6State						:E_Station; 					// Stan pracy podajnika platynek			
	eWeight6RunningState				:E_WeightState; 				// Stan pracy podajnika platynek
	fbWeight6State						:FB_State;					

	(*No nowej wagi*)
	(*wejścia*)
	InWeight6Value 						AT %I*: DINT;			// Wartość wagi
	IbWeight6Overrange 					AT %I*: BOOL;						
	IbWeight6DataInvalid 				AT %I*: BOOL;		
	IbWeight6Error 						AT %I*: BOOL;	
	IbWeight6CalibrationInProgress 		AT %I*: BOOL;
	IbWeight6SteadyState 				AT %I*: BOOL;
	IbWeight6SyncError 					AT %I*: BOOL;
	(*wyjścia*)
	QbWeight6StartCalibration 			AT %Q*: BOOL;
	QbWeight6DisableCalibration 		AT %Q*: BOOL;
	QbWeight6InputFreeze 				AT %Q*: BOOL;
	QbWeight6SampleMode 				AT %Q*: BOOL;
	QbWeight6Tara 						AT %Q*: BOOL;

	(*Ostrzezenia*)
	bWeight6Warning1					:BOOL; // 
	tonWeight6Tare						:TON;		
	
(******** Dozowanie dwufazowe******)		
	
	//Czujniki optyczne przed i za wagą
	fbFilterWeight1: FB_FilterEx;
	fbFilterWeight2: FB_FilterEx;
	fbFilterWeight3: FB_FilterEx;
	fbFilterWeight4: FB_FilterEx;
	fbFilterWeight5: FB_FilterEx;(****** dodane 07.04.2022 przy dodzowniu dwufazowym	**)
	fbFilterWeight6: FB_FilterEx;(****** dodane 07.04.2022 przy dodzowniu dwufazowym	**)

	rFilteredWeight1Value: REAL;
	rFilteredWeight2Value: REAL;
	rFilteredWeight3Value: REAL;
	rFilteredWeight4Value: REAL;
	rFilteredWeight5Value: REAL;(****** dodane 07.04.2022 przy dodzowniu dwufazowym	**)
	rFilteredWeight6Value: REAL;(****** dodane 07.04.2022 przy dodzowniu dwufazowym	**)
	
	//Damian dodane 2 fazy
	fbWeightStation2Phase							: FB_WeightStation;	
	eWeightStation2PhaseState						: E_Station;
	eWeightStation2PhaseRunningState				: E_WeightLiftStationState;
	
	//Dodane Przez Mikołaja
	fbWeightStation									: FB_WeightStation;
	eWeightStationState								: E_Station;
	eWeightStationRunningState						: E_WeightLiftStationState;
	
	IbWeight1ActuatorSensorUp			AT %I*		: BOOL;							//Czujnik podnoszenia Waga 1
	IbWeight2ActuatorSensorUp			AT %I*		: BOOL;							//Czujnik podnoszenia Waga 2
	IbWeight3ActuatorSensorUp			AT %I*		: BOOL;							//Czujnik podnoszenia Waga 3
	IbWeight4ActuatorSensorUp			AT %I*		: BOOL;							//Czujnik podnoszenia Waga 4
	IbWeight5ActuatorSensorUp			AT %I*		: BOOL;							//Czujnik podnoszenia Waga 5 
	IbWeight6ActuatorSensorUp			AT %I*		: BOOL;							//Czujnik podnoszenia Waga 6 
		
	QbWeight1Actuator								: BOOL;							//Podnoszenie Waga 1
    QbWeight2Actuator								: BOOL;							//Podnoszenie Waga 2
	QbWeight3Actuator								: BOOL;							//Podnoszenie Waga 3
	QbWeight4Actuator								: BOOL;							//Podnoszenie Waga 4	                                    		
	QbWeight5Actuator								: BOOL;							//Podnoszenie Waga 5 (2faza)	                                    		
	QbWeight6Actuator								: BOOL;							//Podnoszenie Waga 6 (2faza)

		
	(*Symulacja czujników*)
	tonIbWeight1ActuatorSensorUp					: TON;	
	tonIbWeight2ActuatorSensorUp					: TON;	
	tonIbWeight3ActuatorSensorUp					: TON;	
	tonIbWeight4ActuatorSensorUp					: TON;	
	tonIbWeight5ActuatorSensorUp					: TON;	
	tonIbWeight6ActuatorSensorUp					: TON;	
	
	tonIbWeight1FormSensor: TON;
	tonIbWeight2FormSensor: TON;
	tonIbWeight3FormSensor: TON;
	tonIbWeight4FormSensor: TON;
	tonIbWeight5FormSensor: TON;
	tonIbWeight6FormSensor: TON;
	
	fbIbWeight1FormBeforeSensor: FB_InputFilter_v2;
	fbIbWeight2FormBeforeSensor: FB_InputFilter_v2;
	fbIbWeight3FormBeforeSensor: FB_InputFilter_v2;
	fbIbWeight4FormBeforeSensor: FB_InputFilter_v2;		
	fbIbWeight5FormBeforeSensor: FB_InputFilter_v2;		
	fbIbWeight6FormBeforeSensor: FB_InputFilter_v2;			
	btemp: BOOL;
	
	//wykresy
	fbTrig1 : R_TRIG;
    fbTrig2 : R_TRIG;
    fbTrig3 : R_TRIG;
    fbTrig4 : R_TRIG;
	tSys : DT;
    tTOD : TOD;
	GetTimeSeconds : INT;
	weightIndex : INT;   // 0..7
    valueY : INT;
	i : INT;
	 
	fbHistory: FB_WeightHistory;
END_VAR


fbWeight1.bIgnoreError:=fbWeight2.bIgnoreError:=fbWeight3.bIgnoreError:=fbWeight4.bIgnoreError:=fbWeight5.bIgnoreError:=fbWeight6.bIgnoreError;

aFilter();
aWeight1();
aWeight2();
aWeight3();
aWeight4();
aWeight5();
aWeight6();
ACT_WeightChartDrawers();
IF NOT bDosingTwoPhases THEN
	ACT_WeightStation();
ELSE
	ACT_WeightStation2Phase();
END_IF

// Czas opóżnienia zbierania próbekFB_EntranceGatesServo
fbWeight1.nWeightingDelay:=fbWeight2.nWeightingDelay:=fbWeight3.nWeightingDelay:=fbWeight4.nWeightingDelay:=530;//530
fbWeight5.nWeightingDelay:=fbWeight6.nWeightingDelay:=750;//było 685

(********* GENEROWANIE STANU STACJI DO WIZKI**********)

fbWeight1State(
	eState															:= eWeight1State , 
	bRun															:= VIS.bWeight1DoWeighting,	
	eWeightRunningState												:= eWeight1RunningState , 
	sStateDesc														=> VIS.sWeight1State,
	iState															=> VIS.iWeight1State	);	

fbWeight2State(
	eState															:= eWeight2State , 
	bRun															:= VIS.bWeight2DoWeighting,	
	eWeightRunningState												:= eWeight2RunningState , 
	sStateDesc														=> VIS.sWeight2State,
	iState															=> VIS.iWeight2State	);	
		
fbWeight3State(
	eState															:= eWeight3State , 
	bRun															:= VIS.bWeight3DoWeighting,	
	eWeightRunningState												:= eWeight3RunningState , 
	sStateDesc														=> VIS.sWeight3State,
	iState															=> VIS.iWeight3State	);	
	
fbWeight4State(
	eState															:= eWeight4State , 
	bRun															:= VIS.bWeight4DoWeighting,	
	eWeightRunningState												:= eWeight4RunningState , 
	sStateDesc														=> VIS.sWeight4State,
	iState															=> VIS.iWeight4State	);	
	
fbWeight5State(
	eState															:= eWeight5State , 
	bRun															:= VIS.bWeight5DoWeighting,	
	eWeightRunningState												:= eWeight5RunningState , 
	sStateDesc														=> VIS.sWeight5State,
	iState															=> VIS.iWeight5State	);	

fbWeight6State(
	eState															:= eWeight6State , 
	bRun															:= VIS.bWeight6DoWeighting,	
	eWeightRunningState												:= eWeight6RunningState , 
	sStateDesc														=> VIS.sWeight6State,
	iState															=> VIS.iWeight6State	);		
	
fbWeightLiftState(
	eState															:= eWeightStationState, 
	bRun															:= VIS.bWeightLiftRun OR bWeightLift2PhaseRun,	
	eWeightLiftRunningState											:= eWeightStationRunningState , 
	sStateDesc														=> VIS.sWeightLiftState,
	iState															=> VIS.iWeightLiftState	);		
	
(***** KONIEC GENEROWANIE STANU STACJI DO WIZKI*******)

(****Ostrzezenia***)
// Waga 1
WeightWarning[0].sDescription										:= 'Wagi | Brak stabilizacji przy pomiarach';
IF (bWeight1Warning1 OR bWeight2Warning1 OR bWeight3Warning1 OR bWeight4Warning1 OR bWeight5Warning1 OR bWeight6Warning1) AND NOT WeightWarning[0].bWarning THEN
	WeightWarning[0].bWarning										:= TRUE;
	
ELSIF NOT bWeight1Warning1 AND WeightWarning[0].bAcknowledge THEN
	WeightWarning[0].bWarning										:= FALSE;
	WeightWarning[0].bAcknowledge									:= FALSE;
	VIS.uliWarningAcknowledge.4 										:= FALSE;
	
ELSIF WeightWarning[0].bAcknowledge THEN
	WeightWarning[0].bAcknowledge									:= TRUE;
END_IF


(********KASOWANIE ROZKAZÓW CYKLI*********)
IF fbWeight1.bCycleDone AND bManualMode THEN
	VIS.bWeight1DoWeighting 												:= FALSE;
END_IF

tonWeight1Tare(IN:=VIS.bWeight1Tare,PT:=T#2S);
IF tonWeight1Tare.Q THEN
	VIS.bWeight1Tare												:= FALSE;
END_IF

IF fbWeight2.bCycleDone AND bManualMode THEN
	VIS.bWeight2DoWeighting 												:= FALSE;
END_IF

tonWeight2Tare(IN:=VIS.bWeight2Tare,PT:=T#2S);
IF tonWeight2Tare.Q THEN
	VIS.bWeight2Tare												:= FALSE;
END_IF

IF fbWeight3.bCycleDone AND bManualMode THEN
	VIS.bWeight3DoWeighting 												:= FALSE;
END_IF

tonWeight3Tare(IN:=VIS.bWeight3Tare,PT:=T#2S);
IF tonWeight3Tare.Q THEN
	VIS.bWeight3Tare												:= FALSE;
END_IF
//
IF fbWeight4.bCycleDone AND bManualMode THEN
	VIS.bWeight4DoWeighting 												:= FALSE;
END_IF

tonWeight4Tare(IN:=VIS.bWeight4Tare,PT:=T#2S);
IF tonWeight4Tare.Q THEN
	VIS.bWeight4Tare												:= FALSE;
END_IF

// Waga 5 (1 stacja przy dwufazie)
IF fbWeight5.bCycleDone AND bManualMode THEN
	VIS.bWeight5DoWeighting 												:= FALSE;
END_IF

tonWeight5Tare(IN:=VIS.bWeight5Tare,PT:=T#2S);
IF tonWeight5Tare.Q THEN
	VIS.bWeight5Tare												:= FALSE;
END_IF

// Waga 6 (1 stacja przy dwufazie)
IF fbWeight6.bCycleDone AND bManualMode THEN
	VIS.bWeight6DoWeighting 												:= FALSE;
END_IF

tonWeight6Tare(IN:=VIS.bWeight6Tare,PT:=T#2S);
IF tonWeight6Tare.Q THEN
	VIS.bWeight6Tare												:= FALSE;
END_IF
(*****KONIEC KASOWANIA ROZKAZÓW CYKLI*****)

(**SYMULACJA CZUJNIKÓW**)
tonIbWeight1ActuatorSensorUp(IN:= QbWeight1Actuator, PT:=T#80MS);
tonIbWeight2ActuatorSensorUp(IN:= QbWeight2Actuator, PT:=T#80MS);
tonIbWeight3ActuatorSensorUp(IN:= QbWeight3Actuator, PT:=T#80MS);
tonIbWeight4ActuatorSensorUp(IN:= QbWeight4Actuator, PT:=T#80MS);
tonIbWeight5ActuatorSensorUp(IN:= QbWeight5Actuator, PT:=T#100MS);
tonIbWeight6ActuatorSensorUp(IN:= QbWeight6Actuator, PT:=T#100MS);

ACTION ACT_WeightChartDrawers:
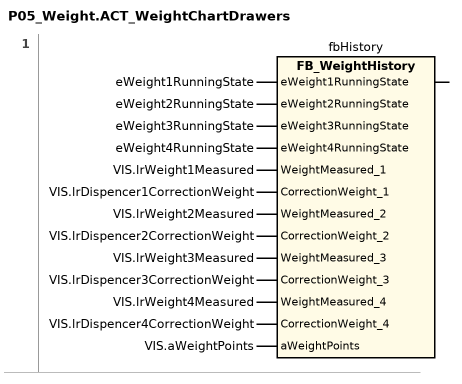
// NETWORK 1
fbHistory(
    eWeight1RunningState := eWeight1RunningState,
    eWeight2RunningState := eWeight2RunningState,
    eWeight3RunningState := eWeight3RunningState,
    eWeight4RunningState := eWeight4RunningState,
    WeightMeasured_1 := VIS.lrWeight1Measured,
    CorrectionWeight_1 := VIS.lrDispencer1CorrectionWeight,
    WeightMeasured_2 := VIS.lrWeight2Measured,
    CorrectionWeight_2 := VIS.lrDispencer2CorrectionWeight,
    WeightMeasured_3 := VIS.lrWeight3Measured,
    CorrectionWeight_3 := VIS.lrDispencer3CorrectionWeight,
    WeightMeasured_4 := VIS.lrWeight4Measured,
    CorrectionWeight_4 := VIS.lrDispencer4CorrectionWeight,
    aWeightPoints := VIS.aWeightPoints); // FB_WeightHistory
END_ACTION

ACTION ACT_WeightStation:
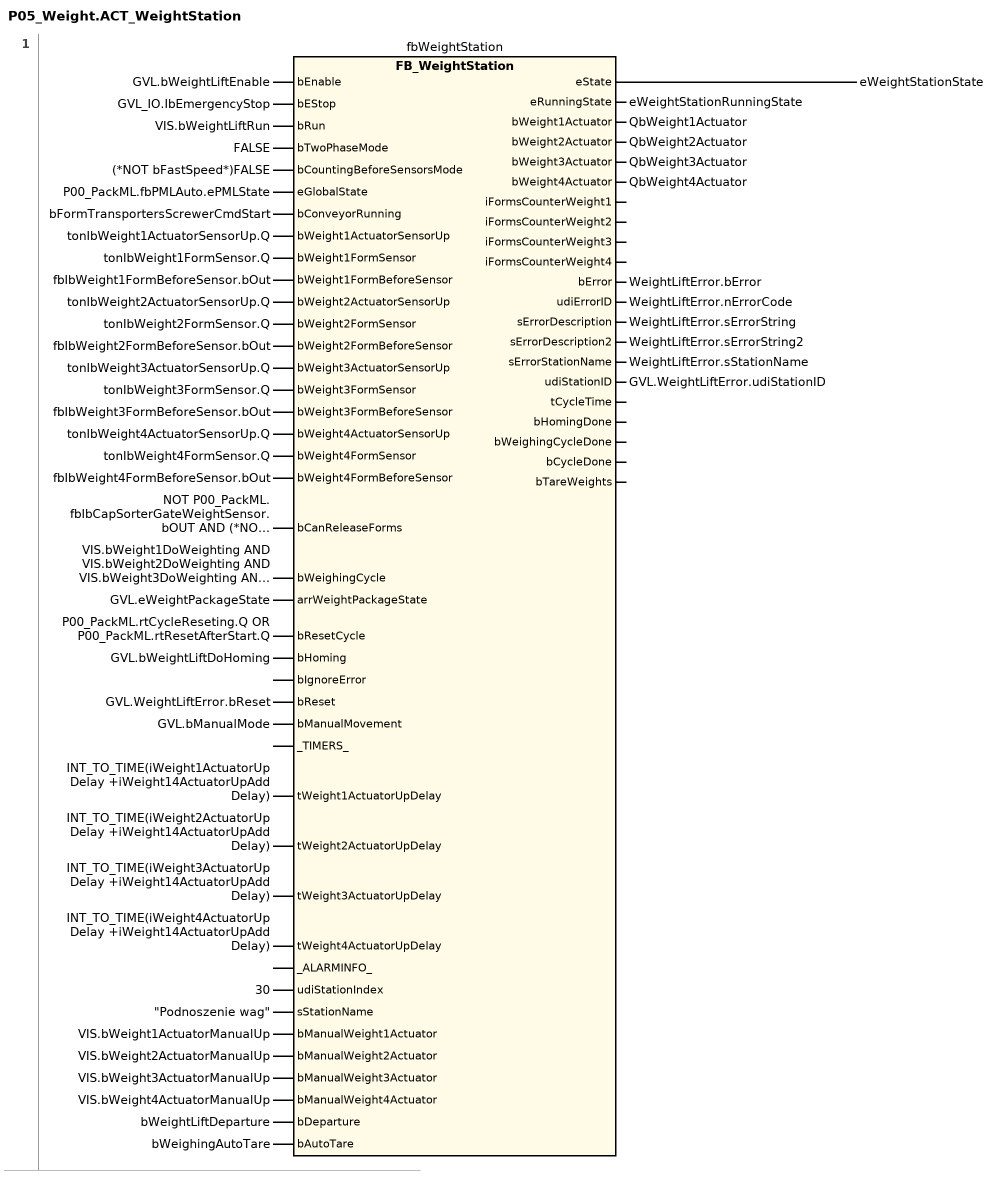
// NETWORK 1
fbWeightStation(
    bEnable := GVL.bWeightLiftEnable,
    bEStop := GVL_IO.IbEmergencyStop,
    bRun := VIS.bWeightLiftRun,
    bTwoPhaseMode := FALSE,
    bCountingBeforeSensorsMode := (*NOT bFastSpeed*)FALSE,
    eGlobalState := P00_PackML.fbPMLAuto.ePMLState,
    bConveyorRunning := bFormTransportersScrewerCmdStart,
    bWeight1ActuatorSensorUp := tonIbWeight1ActuatorSensorUp.Q,
    bWeight1FormSensor := tonIbWeight1FormSensor.Q,
    bWeight1FormBeforeSensor := fbIbWeight1FormBeforeSensor.bOut,
    bWeight2ActuatorSensorUp := tonIbWeight2ActuatorSensorUp.Q,
    bWeight2FormSensor := tonIbWeight2FormSensor.Q,
    bWeight2FormBeforeSensor := fbIbWeight2FormBeforeSensor.bOut,
    bWeight3ActuatorSensorUp := tonIbWeight3ActuatorSensorUp.Q,
    bWeight3FormSensor := tonIbWeight3FormSensor.Q,
    bWeight3FormBeforeSensor := fbIbWeight3FormBeforeSensor.bOut,
    bWeight4ActuatorSensorUp := tonIbWeight4ActuatorSensorUp.Q,
    bWeight4FormSensor := tonIbWeight4FormSensor.Q,
    bWeight4FormBeforeSensor := fbIbWeight4FormBeforeSensor.bOut,
    bCanReleaseForms := NOT P00_PackML.fbIbCapSorterGateWeightSensor.bOUT AND (*NOT P00_PackML.fbIbCapCorrectCheckFormSensor.bOUT AND zalezy od ilosci formatek*)  NOT bWeight1234ReleaseBlock,
    bWeighingCycle := VIS.bWeight1DoWeighting AND VIS.bWeight2DoWeighting AND VIS.bWeight3DoWeighting AND VIS.bWeight4DoWeighting,
    arrWeightPackageState := GVL.eWeightPackageState,
    bResetCycle := P00_PackML.rtCycleReseting.Q OR P00_PackML.rtResetAfterStart.Q,
    bHoming := GVL.bWeightLiftDoHoming,
    bReset := GVL.WeightLiftError.bReset,
    bManualMovement := GVL.bManualMode,
    tWeight1ActuatorUpDelay := INT_TO_TIME(iWeight1ActuatorUpDelay +iWeight14ActuatorUpAddDelay),
    tWeight2ActuatorUpDelay := INT_TO_TIME(iWeight2ActuatorUpDelay +iWeight14ActuatorUpAddDelay),
    tWeight3ActuatorUpDelay := INT_TO_TIME(iWeight3ActuatorUpDelay +iWeight14ActuatorUpAddDelay),
    tWeight4ActuatorUpDelay := INT_TO_TIME(iWeight4ActuatorUpDelay +iWeight14ActuatorUpAddDelay),
    udiStationIndex := 30,
    sStationName := "Podnoszenie wag",
    bManualWeight1Actuator := VIS.bWeight1ActuatorManualUp,
    bManualWeight2Actuator := VIS.bWeight2ActuatorManualUp,
    bManualWeight3Actuator := VIS.bWeight3ActuatorManualUp,
    bManualWeight4Actuator := VIS.bWeight4ActuatorManualUp,
    bDeparture := bWeightLiftDeparture,
    bAutoTare := bWeighingAutoTare,
    eRunningState => eWeightStationRunningState,
    bWeight1Actuator => QbWeight1Actuator,
    bWeight2Actuator => QbWeight2Actuator,
    bWeight3Actuator => QbWeight3Actuator,
    bWeight4Actuator => QbWeight4Actuator,
    bError => WeightLiftError.bError,
    udiErrorID => WeightLiftError.nErrorCode,
    sErrorDescription => WeightLiftError.sErrorString,
    sErrorDescription2 => WeightLiftError.sErrorString2,
    sErrorStationName => WeightLiftError.sStationName,
    udiStationID => GVL.WeightLiftError.udiStationID); // FB_WeightStation
eWeightStationState := fbWeightStation.eState;
END_ACTION

ACTION ACT_WeightStation2Phase:
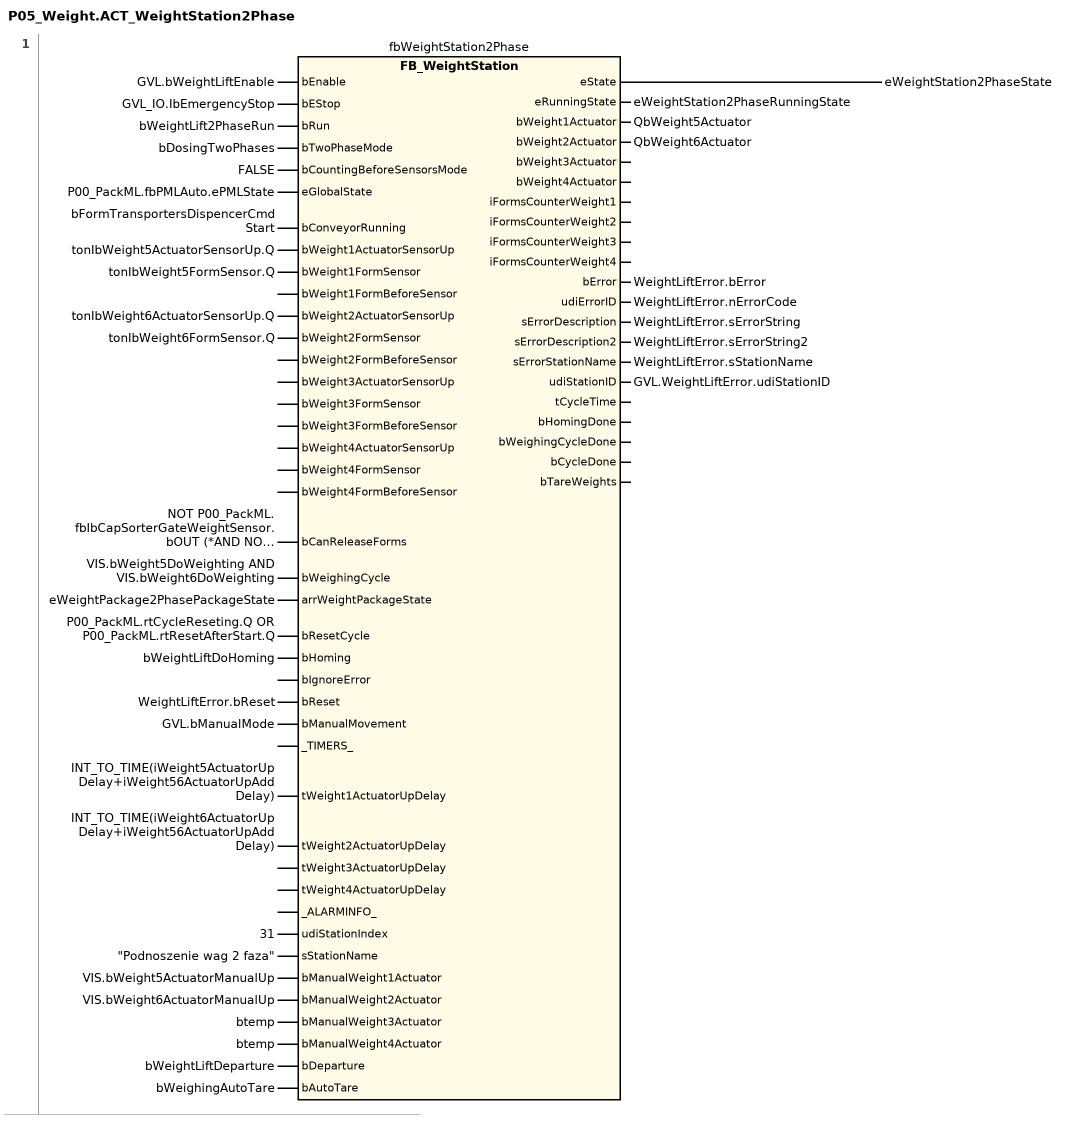
// NETWORK 1
fbWeightStation2Phase(
    bEnable := GVL.bWeightLiftEnable,
    bEStop := GVL_IO.IbEmergencyStop,
    bRun := bWeightLift2PhaseRun,
    bTwoPhaseMode := bDosingTwoPhases,
    bCountingBeforeSensorsMode := FALSE,
    eGlobalState := P00_PackML.fbPMLAuto.ePMLState,
    bConveyorRunning := bFormTransportersDispencerCmdStart,
    bWeight1ActuatorSensorUp := tonIbWeight5ActuatorSensorUp.Q,
    bWeight1FormSensor := tonIbWeight5FormSensor.Q,
    bWeight2ActuatorSensorUp := tonIbWeight6ActuatorSensorUp.Q,
    bWeight2FormSensor := tonIbWeight6FormSensor.Q,
    bCanReleaseForms := NOT P00_PackML.fbIbCapSorterGateWeightSensor.bOUT (*AND NOT P00_PackML.fbIbCapCorrectCheckFormSensor.bOUT*)  AND NOT bWeight56ReleaseBlock,
    bWeighingCycle := VIS.bWeight5DoWeighting AND VIS.bWeight6DoWeighting,
    arrWeightPackageState := eWeightPackage2PhasePackageState,
    bResetCycle := P00_PackML.rtCycleReseting.Q OR P00_PackML.rtResetAfterStart.Q,
    bHoming := bWeightLiftDoHoming,
    bReset := WeightLiftError.bReset,
    bManualMovement := GVL.bManualMode,
    tWeight1ActuatorUpDelay := INT_TO_TIME(iWeight5ActuatorUpDelay+iWeight56ActuatorUpAddDelay),
    tWeight2ActuatorUpDelay := INT_TO_TIME(iWeight6ActuatorUpDelay+iWeight56ActuatorUpAddDelay),
    udiStationIndex := 31,
    sStationName := "Podnoszenie wag 2 faza",
    bManualWeight1Actuator := VIS.bWeight5ActuatorManualUp,
    bManualWeight2Actuator := VIS.bWeight6ActuatorManualUp,
    bManualWeight3Actuator := btemp,
    bManualWeight4Actuator := btemp,
    bDeparture := bWeightLiftDeparture,
    bAutoTare := bWeighingAutoTare,
    eRunningState => eWeightStation2PhaseRunningState,
    bWeight1Actuator => QbWeight5Actuator,
    bWeight2Actuator => QbWeight6Actuator,
    bError => WeightLiftError.bError,
    udiErrorID => WeightLiftError.nErrorCode,
    sErrorDescription => WeightLiftError.sErrorString,
    sErrorDescription2 => WeightLiftError.sErrorString2,
    sErrorStationName => WeightLiftError.sStationName,
    udiStationID => GVL.WeightLiftError.udiStationID); // FB_WeightStation
eWeightStation2PhaseState := fbWeightStation2Phase.eState;
END_ACTION

ACTION aFilter:
fbFilterWeight1(
				rIn:=				DINT_TO_REAL(InWeight1Value), 
				tTimeConstant:= 	T#25MS, //bylo 25
				rOut=>				rFilteredWeight1Value);
							
